    /// <summary>FT-04</summary>
	{attribute 'OPC.UA.DA' := '1'}  				                
	{attribute 'OPC.UA.DA.Access' := '1'}  					                
	product_condenser_pump_outlet_liquid_flow							: REAL;
    /// <summary>FT-04</summary>
	{attribute 'OPC.UA.DA' := '1'}  				                
	{attribute 'OPC.UA.DA.Access' := '1'}  				                
	product_condenser_pump_outlet_liquid_flow_error				AT %I*	: BOOL;
    /// <summary>product condenser pump liquid flow</summary>
	FT_04														AT %I*	: INT;
	
    /// <summary>FT-05</summary>
	{attribute 'OPC.UA.DA' := '1'}  				                
	{attribute 'OPC.UA.DA.Access' := '1'}  					                
	tap_water_to_boiler_flow											: REAL;
	/// <summary>FT-05</summary>
	{attribute 'OPC.UA.DA' := '1'}  				                
	{attribute 'OPC.UA.DA.Access' := '1'}  					                
	tap_water_to_boiler_flow_total										: REAL;
	/// <summary>FT-05</summary>
	{attribute 'OPC.UA.DA' := '1'}  				                					                
	tap_water_to_boiler_flow_total_enable								: BOOL;
    /// <summary>FT-05</summary>
	{attribute 'OPC.UA.DA' := '1'}  				                
	{attribute 'OPC.UA.DA.Access' := '1'}  				                
	tap_water_to_boiler_flow_error								AT %I*	: BOOL;
    /// <summary>tap water to boiler flow</summary>
	FT_05														AT %I*	: INT;

    /// <summary>FT-06</summary>
	{attribute 'OPC.UA.DA' := '1'}  				                
	{attribute 'OPC.UA.DA.Access' := '1'}  					                
	steam_header_flow													: REAL;
	{attribute 'OPC.UA.DA' := '1'}  				                
	{attribute 'OPC.UA.DA.Access' := '1'}
	steam_header_volume  												: REAL;
	 /// <summary>FT-06</summary>
	{attribute 'OPC.UA.DA' := '1'}  				                
	{attribute 'OPC.UA.DA.Access' := '1'}
	steam_header_volume_total 											: REAL;
	  /// <summary>FT-06</summary>
	{attribute 'OPC.UA.DA' := '1'} 
	steam_header_volume_total_enable 									: BOOL;
    /// <summary>FT-06</summary>
	{attribute 'OPC.UA.DA' := '1'}  				                
	{attribute 'OPC.UA.DA.Access' := '1'}  				                
	steam_header_flow_error										AT %I*	: BOOL;
    /// <summary>steam header flow</summary>
	FT_06														AT %I*	: INT;

    /// <summary>FT-07</summary>
	{attribute 'OPC.UA.DA' := '1'}  				                
	{attribute 'OPC.UA.DA.Access' := '1'}  					                
	condensate_collection_tank_flow										: REAL;
    /// <summary>FT-07</summary>
	{attribute 'OPC.UA.DA' := '1'}  				                
	{attribute 'OPC.UA.DA.Access' := '1'}  				                
	condensate_collection_tank_flow_error						AT %I*	: BOOL;
    /// <summary>condensate collection tank flow</summary>
	FT_07														AT %I*	: INT;

    /// <summary>AT-08</summary>
	{attribute 'OPC.UA.DA' := '1'}  				                
	{attribute 'OPC.UA.DA.Access' := '1'}  				                
	weather_wind_speed													: REAL;
    /// <summary>AT-08</summary>                        
	{attribute 'OPC.UA.DA' := '1'}  				                
	{attribute 'OPC.UA.DA.Access' := '1'}  				            
	weather_wind_speed_error									AT %I*	: BOOL;
    /// <summary>weather wind speed</summary>
	AT_08														AT %I*	: INT;

    /// <summary>LT-01</summary>
	{attribute 'OPC.UA.DA' := '1'}  				                
	{attribute 'OPC.UA.DA.Access' := '1'}  					                
	product_condensate_drum_level										: REAL;
    /// <summary>LT-01</summary>
	{attribute 'OPC.UA.DA' := '1'}  				                
	{attribute 'OPC.UA.DA.Access' := '1'}  				                
	product_condensate_drum_level_error							AT %I*	: BOOL;
    /// <summary>product condensate drum level</summary>
	LT_01														AT %I*	: INT;

    /// <summary>LT-02</summary>
	{attribute 'OPC.UA.DA' := '1'}  				                
	{attribute 'OPC.UA.DA.Access' := '1'}  					                
	condensate_collection_tank_level									: REAL;
    /// <summary>LT-02</summary>
	{attribute 'OPC.UA.DA' := '1'}  				                
	{attribute 'OPC.UA.DA.Access' := '1'}  				                
	condensate_collection_tank_level_error						AT %I*	: BOOL;
    /// <summary>condensate collection tank flow</summary>
	LT_02														AT %I*	: INT;

    /// <summary>PT-01</summary>
	{attribute 'OPC.UA.DA' := '1'}  				                
	{attribute 'OPC.UA.DA.Access' := '1'}  				                
	dead_air_line_pres													: REAL;
    /// <summary>PT-01</summary>
	{attribute 'OPC.UA.DA' := '1'}  				                
	{attribute 'OPC.UA.DA.Access' := '1'}  				                
	dead_air_line_pres_error									AT %I*	: BOOL;
    /// <summary>dead air line pres</summary>
	PT_01														AT %I*	: INT;
	
    /// <summary>PT-02</summary>
	{attribute 'OPC.UA.DA' := '1'}  				                
	{attribute 'OPC.UA.DA.Access' := '1'}  				                
	purge_product_line_pres												: REAL;
    /// <summary>PT-02</summary>
	{attribute 'OPC.UA.DA' := '1'}  				                
	{attribute 'OPC.UA.DA.Access' := '1'}  				                
	purge_product_line_pres_error								AT %I*	: BOOL;
    /// <summary>product line pres</summary>
	PT_02														AT %I*	: INT;

    /// <summary>PT-03</summary>
	{attribute 'OPC.UA.DA' := '1'}  				                
	{attribute 'OPC.UA.DA.Access' := '1'}  				                
	pre_condenser_line_pres												: REAL;
    /// <summary>PT-03</summary>
	{attribute 'OPC.UA.DA' := '1'}  				                
	{attribute 'OPC.UA.DA.Access' := '1'}  				                
	pre_condenser_line_pres_error								AT %I*	: BOOL;
    /// <summary>pre condenser line pres</summary>
	PT_03														AT %I*	: INT;

    /// <summary>PT-04</summary>
	{attribute 'OPC.UA.DA' := '1'}  				                
	{attribute 'OPC.UA.DA.Access' := '1'}  				                
	post_condenser_line_pres											: REAL;
    /// <summary>PT-04</summary>
	{attribute 'OPC.UA.DA' := '1'}  				                
	{attribute 'OPC.UA.DA.Access' := '1'}  				                
	post_condenser_line_pres_error								AT %I*	: BOOL;
    /// <summary>post condenser line pres</summary>
	PT_04														AT %I*	: INT;

    /// <summary>PT-05</summary>
	{attribute 'OPC.UA.DA' := '1'}  				                
	{attribute 'OPC.UA.DA.Access' := '1'}  				                
	product_vacuum_pres													: REAL;
    /// <summary>PT-05</summary>
	{attribute 'OPC.UA.DA' := '1'}  				                
	{attribute 'OPC.UA.DA.Access' := '1'}  				                
	product_vacuum_pres_error									AT %I*	: BOOL;
    /// <summary>product vacuum pres</summary>
	PT_05														AT %I*	: INT;

    /// <summary>P02-PT-01</summary>
	{attribute 'OPC.UA.DA' := '1'}  				                
	{attribute 'OPC.UA.DA.Access' := '1'}  				                
	product_vacuum_inlet_pres											: REAL;
    /// <summary>P02-PT-01</summary>
	{attribute 'OPC.UA.DA' := '1'}  				                
	{attribute 'OPC.UA.DA.Access' := '1'}  				                
	product_vacuum_inlet_pres_error								AT %I*	: BOOL;
	
	/// <summary>PT-06</summary>
	{attribute 'OPC.UA.DA' := '1'}  				                
	{attribute 'OPC.UA.DA.Access' := '1'}  				                
	product_outlet_pres													: REAL;
    /// <summary>PT-06</summary>
	{attribute 'OPC.UA.DA' := '1'}  				                
	{attribute 'OPC.UA.DA.Access' := '1'}  				                
	product_outlet_pres_error									AT %I*	: BOOL;
    /// <summary>product outlet pres</summary>
	PT_06														AT %I*	: INT;

    /// <summary>PT-07</summary>
	{attribute 'OPC.UA.DA' := '1'}  				                
	{attribute 'OPC.UA.DA.Access' := '1'}  				                
	boiler_outlet_pres													: REAL;
    /// <summary>PT-07</summary>
	{attribute 'OPC.UA.DA' := '1'}  				                
	{attribute 'OPC.UA.DA.Access' := '1'}  				                
	boiler_outlet_pres_error									AT %I*	: BOOL;
    /// <summary>boiler outlet pres</summary>
	PT_07														AT %I*	: INT;

    /// <summary>PT-08</summary>
	{attribute 'OPC.UA.DA' := '1'}  				                
	{attribute 'OPC.UA.DA.Access' := '1'}  				                
	instrument_air_comp_pres											: REAL;
    /// <summary>PT-08</summary>
	{attribute 'OPC.UA.DA' := '1'}  				                
	{attribute 'OPC.UA.DA.Access' := '1'}  				                
	instrument_air_comp_pres_error								AT %I*	: BOOL;
    /// <summary>instrument air comp pres</summary>
	PT_08														AT %I*	: INT;

    /// <summary>PT-09</summary>
	{attribute 'OPC.UA.DA' := '1'}  				                
	{attribute 'OPC.UA.DA.Access' := '1'}  				                
	weather_pres														: REAL;
    /// <summary>PT-09</summary>                        
	{attribute 'OPC.UA.DA' := '1'}  				                
	{attribute 'OPC.UA.DA.Access' := '1'}  				            
	weather_pres_error											AT %I*	: BOOL;
    /// <summary>weather pres</summary>
	PT_09														AT %I*	: INT;


    /// <summary>TT-01</summary>
	{attribute 'OPC.UA.DA' := '1'}  				                
	{attribute 'OPC.UA.DA.Access' := '1'}  				                
	purge_product_line_temp												: REAL;
    /// <summary>TT-01</summary>
	{attribute 'OPC.UA.DA' := '1'}  				                
	{attribute 'OPC.UA.DA.Access' := '1'}  				                
	purge_product_line_temp_error								AT %I*	: BOOL;
    /// <summary>purge product line temp</summary>
	TT_01														AT %I*	: INT;

    /// <summary>TT-02</summary>
	{attribute 'OPC.UA.DA' := '1'}  				                
	{attribute 'OPC.UA.DA.Access' := '1'}  				                
	pre_condenser_line_temp												: REAL;
    /// <summary>TT-02</summary>
	{attribute 'OPC.UA.DA' := '1'}  				                
	{attribute 'OPC.UA.DA.Access' := '1'}  				                
	pre_condenser_line_temp_error								AT %I*	: BOOL;
    /// <summary>pre condenser line temp</summary>
	TT_02														AT %I*	: INT;

    /// <summary>TT-03</summary>
	{attribute 'OPC.UA.DA' := '1'}  				                
	{attribute 'OPC.UA.DA.Access' := '1'}  				                
	post_condenser_line_temp												: REAL;
    /// <summary>TT-03</summary>
	{attribute 'OPC.UA.DA' := '1'}  				                
	{attribute 'OPC.UA.DA.Access' := '1'}  				                
	post_condenser_line_temp_error								AT %I*	: BOOL;
    /// <summary>purge product line temp</summary>
	TT_03														AT %I*	: INT;

    /// <summary>TT-04</summary>
	{attribute 'OPC.UA.DA' := '1'}  				                
	{attribute 'OPC.UA.DA.Access' := '1'}  				                
	product_outlet_temp													: REAL;
    /// <summary>TT-04</summary>
	{attribute 'OPC.UA.DA' := '1'}  				                
	{attribute 'OPC.UA.DA.Access' := '1'}  				                
	product_outlet_temp_error									AT %I*	: BOOL;
    /// <summary>product outlet temp</summary>
	TT_04														AT %I*	: INT;

    /// <summary>TT-05</summary>
	{attribute 'OPC.UA.DA' := '1'}  				                
	{attribute 'OPC.UA.DA.Access' := '1'}  				                
	product_condenser_pump_outlet_temp									: REAL;
    /// <summary>TT-05</summary>
	{attribute 'OPC.UA.DA' := '1'}  				                
	{attribute 'OPC.UA.DA.Access' := '1'}  				                
	product_condenser_pump_outlet_temp_error					AT %I*	: BOOL;
    /// <summary>product condenser pump outlet temp</summary>
	TT_05														AT %I*	: INT;

    /// <summary>TT-06</summary>
	{attribute 'OPC.UA.DA' := '1'}  				                
	{attribute 'OPC.UA.DA.Access' := '1'}  				                
	boiler_outlet_temp													: REAL;
    /// <summary>TT-06</summary>
	{attribute 'OPC.UA.DA' := '1'}  				                
	{attribute 'OPC.UA.DA.Access' := '1'}  				                
	boiler_outlet_temp_error									AT %I*	: BOOL;
    /// <summary>boiler outlet temp</summary>
	TT_06														AT %I*	: INT;

    /// <summary>TT-07</summary>
	{attribute 'OPC.UA.DA' := '1'}  				                
	{attribute 'OPC.UA.DA.Access' := '1'}  				                
	condensate_collection_tank_temp										: REAL;
    /// <summary>TT-07</summary>
	{attribute 'OPC.UA.DA' := '1'}  				                
	{attribute 'OPC.UA.DA.Access' := '1'}  				                
	condensate_collection_tank_temp_error						AT %I*	: BOOL;
    /// <summary>condensate collection tank temp</summary>
	TT_07														AT %I*	: INT;

    /// <summary>TT-08</summary>
	{attribute 'OPC.UA.DA' := '1'}  				                
	{attribute 'OPC.UA.DA.Access' := '1'}  				                
	condensate_collection_tank_outlet_line_temp							: REAL;
    /// <summary>TT-08</summary>
	{attribute 'OPC.UA.DA' := '1'}  				                
	{attribute 'OPC.UA.DA.Access' := '1'}  				                
	condensate_collection_tank_outlet_line_temp_error			AT %I*	: BOOL;
    /// <summary>condensate collection tank outlet temp</summary>
	TT_08														AT %I*	: INT;

    /// <summary>TT-09</summary>
	{attribute 'OPC.UA.DA' := '1'}  				                
	{attribute 'OPC.UA.DA.Access' := '1'}  				                
	instrument_air_comp_temp											: REAL;
    /// <summary>TT-09</summary>
	{attribute 'OPC.UA.DA' := '1'}  				                
	{attribute 'OPC.UA.DA.Access' := '1'}  				                
	instrument_air_comp_temp_error								AT %I*	: BOOL;
    /// <summary>instrument air comp temp</summary>
	TT_09														AT %I*	: INT;

    /// <summary>TT-10</summary>
	{attribute 'OPC.UA.DA' := '1'}  				                
	{attribute 'OPC.UA.DA.Access' := '1'}  				                
	weather_temp														: REAL;
    /// <summary>TT-10</summary>
	{attribute 'OPC.UA.DA' := '1'}  				                
	{attribute 'OPC.UA.DA.Access' := '1'}  				                
	weather_temp_error											AT %I*	: BOOL;
    /// <summary>instrument air comp temp</summary>
	TT_10														AT %I*	: INT;


    /// <summary>NT-01</summary>
	{attribute 'OPC.UA.DA' := '1'}  				                
	{attribute 'OPC.UA.DA.Access' := '1'}  				                
	weather_noise_level													: REAL;
    /// <summary>NT-01</summary>
	{attribute 'OPC.UA.DA' := '1'}  				                
	{attribute 'OPC.UA.DA.Access' := '1'}  				                
	weather_noise_level_error									AT %I*	: BOOL;
    /// <summary>weather noise level</summary>
	NT_01														AT %I*	: INT;

	
    /// <summary>WDT-01</summary>
	{attribute 'OPC.UA.DA' := '1'}  				                
	{attribute 'OPC.UA.DA.Access' := '1'}  				                
	weather_wind_direction												: REAL;
    /// <summary>WDT-01</summary>
	{attribute 'OPC.UA.DA' := '1'}  				                
	{attribute 'OPC.UA.DA.Access' := '1'}  				                
	weather_wind_direction_error								AT %I*	: BOOL;
    /// <summary>weather wind direction</summary>
	WDT_01														AT %I*	: INT;

	
    /// <summary>XV-01</summary>
	{attribute 'OPC.UA.DA' := '1'}  				                
	cooling_line_pre_condenser_valve									: BOOL;
    /// <summary>XV-01</summary>
	{attribute 'OPC.UA.DA' := '1'}  				                
	{attribute 'OPC.UA.DA.Access' := '1'}  				                
	cooling_line_pre_condenser_valve_open_cmd_status					: BOOL;
    /// <summary>XV-01</summary>
	{attribute 'OPC.UA.DA' := '1'}  				                
	{attribute 'OPC.UA.DA.Access' := '1'}  				                
	cooling_line_pre_condenser_valve_open						AT %I*	: BOOL;
    /// <summary>XV-01</summary>
	{attribute 'OPC.UA.DA' := '1'}  				                
	{attribute 'OPC.UA.DA.Access' := '1'}  				                
	cooling_line_pre_condenser_valve_closed						AT %I*	: BOOL;
    /// <summary>cooling line pre condenser valve</summary>
	XV_01														AT %Q*	: BOOL;
	
    /// <summary>XV-02</summary>
	{attribute 'OPC.UA.DA' := '1'}  				                
	purge_product_pre_condenser_valve									: BOOL;
    /// <summary>XV-02</summary>
	{attribute 'OPC.UA.DA' := '1'}  				                
	{attribute 'OPC.UA.DA.Access' := '1'}  				                
	purge_product_pre_condenser_valve_open_cmd_status					: BOOL;
    /// <summary>XV-02</summary>
	{attribute 'OPC.UA.DA' := '1'}  				                
	{attribute 'OPC.UA.DA.Access' := '1'}  				                
	purge_product_pre_condenser_valve_open						AT %I*	: BOOL;
    /// <summary>XV-02</summary>
	{attribute 'OPC.UA.DA' := '1'}  				                
	{attribute 'OPC.UA.DA.Access' := '1'}  				                
	purge_product_pre_condenser_valve_closed					AT %I*	: BOOL;
    /// <summary>purge product pre condenser valve</summary>
	XV_02														AT %Q*	: BOOL;
	
    /// <summary>XV-03</summary>
	{attribute 'OPC.UA.DA' := '1'}  				                
	product_vacuum_pump_isolation_valve									: BOOL;
    /// <summary>XV-03</summary>
	{attribute 'OPC.UA.DA' := '1'}  				                
	{attribute 'OPC.UA.DA.Access' := '1'}  				                
	product_vacuum_pump_isolation_valve_open_cmd_status					: BOOL;
    /// <summary>XV-03</summary>
	{attribute 'OPC.UA.DA' := '1'}  				                
	{attribute 'OPC.UA.DA.Access' := '1'}  				                
	product_vacuum_pump_isolation_valve_open					AT %I*	: BOOL;
    /// <summary>XV-03</summary>
	{attribute 'OPC.UA.DA' := '1'}  				                
	{attribute 'OPC.UA.DA.Access' := '1'}  				                
	product_vacuum_pump_isolation_valve_closed					AT %I*	: BOOL;
    /// <summary>product vacuum pump isolation valve</summary>
	XV_03														AT %Q*	: BOOL;
	
    /// <summary>XV-04</summary>
	{attribute 'OPC.UA.DA' := '1'}  				                
	product_vacuum_bypass_valve											: BOOL;
    /// <summary>XV-04</summary>
	{attribute 'OPC.UA.DA' := '1'}  				                
	{attribute 'OPC.UA.DA.Access' := '1'}  				                
	product_vacuum_bypass_valve_open_cmd_status							: BOOL;
    /// <summary>XV-04</summary>
	{attribute 'OPC.UA.DA' := '1'}  				                
	{attribute 'OPC.UA.DA.Access' := '1'}  				                
	product_vacuum_bypass_valve_open							AT %I*	: BOOL;
    /// <summary>XV-04</summary>
	{attribute 'OPC.UA.DA' := '1'}  				                
	{attribute 'OPC.UA.DA.Access' := '1'}  				                
	product_vacuum_bypass_valve_closed							AT %I*	: BOOL;
    /// <summary>product vacuum bypass valve</summary>
	XV_04														AT %Q*	: BOOL;
	
    /// <summary>XV-05</summary>
	{attribute 'OPC.UA.DA' := '1'}  				                
	product_vacuum_outlet_isolation_valve								: BOOL;
    /// <summary>XV-05</summary>
	{attribute 'OPC.UA.DA' := '1'}  				                
	{attribute 'OPC.UA.DA.Access' := '1'}  				                
	product_vacuum_outlet_isolation_valve_open_cmd_status				: BOOL;
    /// <summary>XV-05</summary>
	{attribute 'OPC.UA.DA' := '1'}  				                
	{attribute 'OPC.UA.DA.Access' := '1'}  				                
	product_vacuum_outlet_isolation_valve_open					AT %I*	: BOOL;
    /// <summary>XV-05</summary>
	{attribute 'OPC.UA.DA' := '1'}  				                
	{attribute 'OPC.UA.DA.Access' := '1'}  				                
	product_vacuum_outlet_isolation_valve_closed				AT %I*	: BOOL;
    /// <summary>product vacuum outlet isolation valve</summary>
	XV_05														AT %Q*	: BOOL;
	
    /// <summary>XV-06</summary>
	{attribute 'OPC.UA.DA' := '1'}  				                
	product_condensate_drain_valve										: BOOL;
    /// <summary>XV-06</summary>
	{attribute 'OPC.UA.DA' := '1'}  				                
	{attribute 'OPC.UA.DA.Access' := '1'}  				                
	product_condensate_drain_valve_open_cmd_status						: BOOL;
    /// <summary>XV-06</summary>
	{attribute 'OPC.UA.DA' := '1'}  				                
	{attribute 'OPC.UA.DA.Access' := '1'}  				                
	product_condensate_drain_valve_open							AT %I*	: BOOL;
    /// <summary>XV-06</summary>
	{attribute 'OPC.UA.DA' := '1'}  				                
	{attribute 'OPC.UA.DA.Access' := '1'}  				                
	product_condensate_drain_valve_closed						AT %I*	: BOOL;
    /// <summary>product condensate drain valve</summary>
	XV_06														AT %Q*	: BOOL;
	
    /// <summary>XV-08</summary>
	{attribute 'OPC.UA.DA' := '1'}  				                
	steam_bypass_valve													: BOOL;
    /// <summary>XV-08</summary>
	{attribute 'OPC.UA.DA' := '1'}  				                
	{attribute 'OPC.UA.DA.Access' := '1'}  				                
	steam_bypass_valve_open_cmd_status									: BOOL;
    /// <summary>XV-08</summary>
	{attribute 'OPC.UA.DA' := '1'}  				                
	{attribute 'OPC.UA.DA.Access' := '1'}  				                
	steam_bypass_valve_open										AT %I*	: BOOL;
    /// <summary>XV-08</summary>
	{attribute 'OPC.UA.DA' := '1'}  				                
	{attribute 'OPC.UA.DA.Access' := '1'}  				                
	steam_bypass_valve_closed									AT %I*	: BOOL;
    /// <summary>steam bypass valve</summary>
	XV_08														AT %Q*	: BOOL;
    
	/// <summary>XV-09</summary>
	{attribute 'OPC.UA.DA' := '1'}  				                
	condensate_collection_tank_pump_outlet_valve						: BOOL;
    /// <summary>XV-09</summary>
	{attribute 'OPC.UA.DA' := '1'}  				                
	{attribute 'OPC.UA.DA.Access' := '1'}  				                
	condensate_collection_tank_pump_outlet_valve_open_cmd_status		: BOOL;
    /// <summary>XV-09</summary>
	{attribute 'OPC.UA.DA' := '1'}  				                
	{attribute 'OPC.UA.DA.Access' := '1'}  				                
	condensate_collection_tank_pump_outlet_valve_open			AT %I*	: BOOL;
    /// <summary>XV-09</summary>
	{attribute 'OPC.UA.DA' := '1'}  				                
	{attribute 'OPC.UA.DA.Access' := '1'}  				                
	condensate_collection_tank_pump_outlet_valve_closed 		AT %I*	: BOOL;
    /// <summary>condensate collection tank pump outlet valve</summary>
	XV_09														AT %Q*	: BOOL;

    /// <summary>PCV-01</summary>
	product_vacuum_backfeed_valve_open									: BOOL;
    /// <summary>PCV-01</summary>
	product_vacuum_backfeed_valve_closed								: BOOL;
    /// <summary>PCV-01</summary>
	{attribute 'OPC.UA.DA' := '1'}  				                
	product_vacuum_backfeed_valve										: REAL;
    /// <summary>PCV-01</summary>
	{attribute 'OPC.UA.DA' := '1'}  				                
	{attribute 'OPC.UA.DA.Access' := '1'}  				                
	product_vacuum_backfeed_valve_position								: REAL;
    /// <summary>PCV-01</summary>
	{attribute 'OPC.UA.DA' := '1'}  				                
	{attribute 'OPC.UA.DA.Access' := '1'}  				                
	product_vacuum_backfeed_valve_position_error				AT %I*	: BOOL;
    /// <summary>product vacuum backfeed valve</summary>
	PCV_01														AT %Q*	: INT;
    /// <summary>product vacuum backfeed valve</summary>
	{attribute 'OPC.UA.DA' := '1'}  				                
	{attribute 'OPC.UA.DA.Access' := '1'}  				                
	PCV_01_position												AT %I*	: INT;
    /// <summary>PCV-01</summary>                  	           
	{attribute 'OPC.UA.DA' := '1'}  				                
	product_vacuum_backfeed_valve_mode									: INT;			
    /// <summary>PCV-01</summary>                  	           
	{attribute 'OPC.UA.DA' := '1'}  				                
	{attribute 'OPC.UA.DA.Access' := '1'}  				                
	product_vacuum_backfeed_valve_current_mode							: INT;			
    /// <summary>PCV-01</summary>                  	           
	product_vacuum_backfeed_valve_kp									: REAL		:= 0.01; 
    /// <summary>PCV-01</summary>                  	           
	product_vacuum_backfeed_valve_ki									: REAL		:= 0.01;
    /// <summary>PCV-01</summary>                  	           
	product_vacuum_backfeed_valve_loop_time								: REAL		:= 2000;
    /// <summary>PCV-01</summary>                  	           
	product_vacuum_backfeed_valve_iband									: REAL		:= 6;
    /// <summary>PCV-01</summary>                  	           
	product_vacuum_backfeed_valve_base									: INT		:= 13110;
    /// <summary>PCV-01</summary>                  	           
	product_vacuum_backfeed_valve_base_adjust							: INT		:= 10;
	
    /// <summary>P-02</summary>
	{attribute 'OPC.UA.DA' := '1'}  				                
	product_vacuum_pump_reset											: BOOL;												// PS 04_17_24 Added for Vacuum Pump FB reset
    /// <summary>P-02</summary>
	{attribute 'OPC.UA.DA' := '1'}  				                
	product_vacuum_pump_vfd_reset										: BOOL;
	  /// <summary>P-02</summary>
	{attribute 'OPC.UA.DA' := '1'}  				                
	product_vacuum_pump_vfd_enable										: BOOL;
    /// <summary>P-02</summary>
	{attribute 'OPC.UA.DA' := '1'}  				                
	{attribute 'OPC.UA.DA.Access' := '1'}  				                
	product_vacuum_pump_vfd_enabled										: BOOL;
    /// <summary>P-02</summary>
	{attribute 'OPC.UA.DA' := '1'}  				                
	{attribute 'OPC.UA.DA.Access' := '1'}  				                
	product_vacuum_pump_vfd_error										: BOOL;
    /// <summary>P-02</summary>
	{attribute 'OPC.UA.DA' := '1'}  				                
	product_vacuum_pump_vfd												: REAL;
    /// <summary>P-02</summary>
	{attribute 'OPC.UA.DA' := '1'}  				                
    /// <summary>P-02</summary>
	product_vacuum_pump_vfd_output										: REAL;
    /// <summary>P-02</summary>
	product_vacuum_pump_vfd_control								AT %Q*	: WORD;
    /// <summary>P-02</summary>
	product_vacuum_pump_vfd_target_vel							AT %Q*	: WORD;
    /// <summary>P-02</summary>
	product_vacuum_pump_vfd_status								AT %I*	: WORD;
    /// <summary>P-02</summary>
	product_vacuum_pump_vfd_velocity							AT %I*	: WORD;

    /// <summary>product_vacuum_pump_pressure</summary>
	P02_PT_01													AT %I*	: INT;
    /// <summary>product_vacuum_pump_cooling_jacket_temp_trip_switch</summary>
	P02_TSH_1													AT %I*	: BOOL;
    /// <summary>product_vacuum_pump_exhaust_temp_trip_switch</summary>
	P02_TSH_2													AT %I*	: BOOL;
    /// <summary>product_vacuum_pump_oil_temp_trip_switch</summary>
	P02_TSH_3													AT %I*	: BOOL;
    /// <summary>product_vacuum_pump_purge_solenoid_valve</summary>
	P02_SVC_1													AT %Q*	: BOOL;
    /// <summary>product_vacuum_pump_seal_purge_valve</summary>
	P02_SVC_3													AT %Q*	: BOOL;
	product_vacuum_pump_error											: INT;
	
	
	  /// <summary>AT-04_pump</summary>
	{attribute 'OPC.UA.DA' := '1'}  				                
	product_co2_chiller_pump											: BOOL;
    /// <summary>AT-04_pump</summary>
	{attribute 'OPC.UA.DA' := '1'}  				                
	{attribute 'OPC.UA.DA.Access' := '1'}  				                
	product_co2_chiller_pump_cmd_status									: BOOL;
    /// <summary>product chiller CO2 pump</summary>
	AT_04_pump													AT %Q*	: BOOL;
    /// <summary>AT-04_chiller</summary>
	{attribute 'OPC.UA.DA' := '1'}  				                
	product_co2_chiller													: BOOL;
    /// <summary>AT-04_chiller</summary>
	{attribute 'OPC.UA.DA' := '1'}  				                
	{attribute 'OPC.UA.DA.Access' := '1'}  				                
	product_co2_chiller_cmd_status											: BOOL;
    /// <summary>productCO2 chiller</summary>
	AT_04_chiller												AT %Q*	: BOOL;
	
	
	
	{attribute 'OPC.UA.DA' := '1'}  				                
	{attribute 'OPC.UA.DA.Access' := '1'}  				                
	l1_current_480														: REAL;
	{attribute 'OPC.UA.DA' := '1'}  				                
	{attribute 'OPC.UA.DA.Access' := '1'}  				                
	l1_current_480_error										AT %I*	: BOOL;
	IT_01														AT %I*	: INT;
	{attribute 'OPC.UA.DA' := '1'}  				                
	{attribute 'OPC.UA.DA.Access' := '1'}  				                
	l2_current_480														: REAL;
	{attribute 'OPC.UA.DA' := '1'}  				                
	{attribute 'OPC.UA.DA.Access' := '1'}  				                
	l2_current_480_error										AT %I*	: BOOL;
	IT_02														AT %I*	: INT;
	{attribute 'OPC.UA.DA' := '1'}  				                
	{attribute 'OPC.UA.DA.Access' := '1'}  				                
	l3_current_480														: REAL;
	{attribute 'OPC.UA.DA' := '1'}  				                
	{attribute 'OPC.UA.DA.Access' := '1'}  				                
	l3_current_480_error										AT %I*	: BOOL;
	IT_03														AT %I*	: INT;
	
	{attribute 'OPC.UA.DA' := '1'}  				                
	{attribute 'OPC.UA.DA.Access' := '1'}  				                
	l1_voltage_480														: REAL;
	{attribute 'OPC.UA.DA' := '1'}  				                
	{attribute 'OPC.UA.DA.Access' := '1'}  				                
	l1_voltage_480_error										AT %I*	: BOOL;
	{attribute 'OPC.UA.DA' := '1'}  				                
	VT_01														AT %I*	: INT;
	{attribute 'OPC.UA.DA' := '1'}  				                
	l2_voltage_480														: REAL;
	{attribute 'OPC.UA.DA' := '1'}  				                
	{attribute 'OPC.UA.DA.Access' := '1'}  				                
	l2_voltage_480_error										AT %I*	: BOOL;
	{attribute 'OPC.UA.DA' := '1'}  				                
	VT_02														AT %I*	: INT;
	{attribute 'OPC.UA.DA' := '1'}  				                
	l3_voltage_480														: REAL;
	{attribute 'OPC.UA.DA' := '1'}  				                
	{attribute 'OPC.UA.DA.Access' := '1'}  				                
	l3_voltage_480_error										AT %I*	: BOOL;
	{attribute 'OPC.UA.DA' := '1'}  				                
	VT_03														AT %I*	: INT;
	
	{attribute 'OPC.UA.DA' := '1'}  				                
	{attribute 'OPC.UA.DA.Access' := '1'}  				                
	l1_current_208														: REAL;
	{attribute 'OPC.UA.DA' := '1'}  				                
	{attribute 'OPC.UA.DA.Access' := '1'}  				                
	l1_current_208_error										AT %I*	: BOOL;
	IT_04														AT %I*	: INT;
	{attribute 'OPC.UA.DA' := '1'}  				                
	{attribute 'OPC.UA.DA.Access' := '1'}  				                
	l2_current_208														: REAL;
	{attribute 'OPC.UA.DA' := '1'}  				                
	{attribute 'OPC.UA.DA.Access' := '1'}  				                
	l2_current_208_error										AT %I*	: BOOL;
	IT_05														AT %I*	: INT;
	{attribute 'OPC.UA.DA' := '1'}  				                
	{attribute 'OPC.UA.DA.Access' := '1'}  				                
	l3_current_208														: REAL;
	{attribute 'OPC.UA.DA' := '1'}  				                
	{attribute 'OPC.UA.DA.Access' := '1'}  				                
	l3_current_208_error										AT %I*	: BOOL;
	IT_06														AT %I*	: INT;
	
	{attribute 'OPC.UA.DA' := '1'}  				                
	{attribute 'OPC.UA.DA.Access' := '1'}  				                
	l1_voltage_208														: REAL;
	{attribute 'OPC.UA.DA' := '1'}  				                
	{attribute 'OPC.UA.DA.Access' := '1'}  				                
	l1_voltage_208_error										AT %I*	: BOOL;
	VT_04														AT %I*	: INT;
	{attribute 'OPC.UA.DA' := '1'}  				                
	{attribute 'OPC.UA.DA.Access' := '1'}  				                
	l2_voltage_208														: REAL;
	{attribute 'OPC.UA.DA' := '1'}  				                
	{attribute 'OPC.UA.DA.Access' := '1'}  				                
	l2_voltage_208_error										AT %I*	: BOOL;
	VT_05														AT %I*	: INT;
	{attribute 'OPC.UA.DA' := '1'}  				                
	{attribute 'OPC.UA.DA.Access' := '1'}  				                
	l3_voltage_208														: REAL;
	{attribute 'OPC.UA.DA' := '1'}  				                
	{attribute 'OPC.UA.DA.Access' := '1'}  				                
	l3_voltage_208_error										AT %I*	: BOOL;
	VT_06														AT %I*	: INT;
	
	{attribute 'OPC.UA.DA' := '1'}  				                
	{attribute 'OPC.UA.DA.Access' := '1'}  				                
	l1_current_boiler													: REAL;
	{attribute 'OPC.UA.DA' := '1'}  				                
	{attribute 'OPC.UA.DA.Access' := '1'}  				                
	l1_current_boiler_error										AT %I*	: BOOL;
	IT_boiler_01												AT %I*	: INT;
	{attribute 'OPC.UA.DA' := '1'}  				                
	{attribute 'OPC.UA.DA.Access' := '1'}  				                
	l2_current_boiler													: REAL;
	{attribute 'OPC.UA.DA' := '1'}  				                
	{attribute 'OPC.UA.DA.Access' := '1'}  				                
	l2_current_boiler_error										AT %I*	: BOOL;
	IT_boiler_02												AT %I*	: INT;
	{attribute 'OPC.UA.DA' := '1'}  				                
	{attribute 'OPC.UA.DA.Access' := '1'}  				                
	l3_current_boiler													: REAL;
	{attribute 'OPC.UA.DA' := '1'}  				                
	{attribute 'OPC.UA.DA.Access' := '1'}  				                
	l3_current_boiler_error										AT %I*	: BOOL;
	IT_boiler_03												AT %I*	: INT;
	
END_VAR

VAR_GLOBAL PERSISTENT
	
	/// SCALING
	
    /// <summary>AT-01</summary>
	{attribute 'OPC.UA.DA' := '1'}  				                
	dead_air_line_co2_low												: REAL;
    /// <summary>AT-01</summary>
	{attribute 'OPC.UA.DA' := '1'}  				                
	dead_air_line_co2_high												: REAL;
    /// <summary>AT-01</summary>
	{attribute 'OPC.UA.DA' := '1'}  				                
	dead_air_line_co2_min												: REAL;
    /// <summary>AT-01</summary>
	{attribute 'OPC.UA.DA' := '1'}  				                
	dead_air_line_co2_offset											: REAL;
	
    /// <summary>AT-02</summary>
	{attribute 'OPC.UA.DA' := '1'}  				                
	product_outlet_co2_low												: REAL;
    /// <summary>AT-02</summary>
	{attribute 'OPC.UA.DA' := '1'}  				                
	product_outlet_co2_high												: REAL;
    /// <summary>AT-02</summary>
	{attribute 'OPC.UA.DA' := '1'}  				                
	product_outlet_co2_min												: REAL;
    /// <summary>AT-02</summary>
	{attribute 'OPC.UA.DA' := '1'}  				                
	product_outlet_co2_offset											: REAL;
	
	/// <summary>AT-02</summary>
	{attribute 'OPC.UA.DA' := '1'}  				                
	product_co2sample_h2o_low											: REAL;
    /// <summary>AT-02</summary>
	{attribute 'OPC.UA.DA' := '1'}  				                
	product_co2sample_h2o_high											: REAL;
    /// <summary>AT-02</summary>
	{attribute 'OPC.UA.DA' := '1'}  				                
	product_co2sample_h2o_min											: REAL;
    /// <summary>AT-02</summary>
	{attribute 'OPC.UA.DA' := '1'}  				                
	product_co2sample_h2o_offset										: REAL;
	
	
    /// <summary>AT-07</summary>
	{attribute 'OPC.UA.DA' := '1'}  				                
	product_outlet_h2o_low												: REAL;
    /// <summary>AT-07</summary>
	{attribute 'OPC.UA.DA' := '1'}  				                
	product_outlet_h2o_high												: REAL;
    /// <summary>AT-07</summary>
	{attribute 'OPC.UA.DA' := '1'}  				                
	product_outlet_h2o_min												: REAL;
    /// <summary>AT-07</summary>
	{attribute 'OPC.UA.DA' := '1'}  				                
	product_outlet_h2o_offset											: REAL;
	
	
	 /// <summary>AT-07</summary>
	{attribute 'OPC.UA.DA' := '1'}  				                
	product_outlet_temperature_low										: REAL;
    /// <summary>AT-07</summary>
	{attribute 'OPC.UA.DA' := '1'}  				                
	product_outlet_temperature_high										: REAL;
    /// <summary>AT-07</summary>
	{attribute 'OPC.UA.DA' := '1'}  				                
	product_outlet_temperature_min										: REAL;
    /// <summary>AT-07</summary>
	{attribute 'OPC.UA.DA' := '1'}  				                
	product_outlet_temperature_offset									: REAL;
	
    /// <summary>AT-03</summary>
	{attribute 'OPC.UA.DA' := '1'}  				                
	product_outlet_o2_low												: REAL;
    /// <summary>AT-03</summary>
	{attribute 'OPC.UA.DA' := '1'}  				                
	product_outlet_o2_high												: REAL;
    /// <summary>AT-03</summary>
	{attribute 'OPC.UA.DA' := '1'}  				                
	product_outlet_o2_min												: REAL;
    /// <summary>AT-03</summary>
	{attribute 'OPC.UA.DA' := '1'}  				                
	product_outlet_o2_offset											: REAL;
	
    /// <summary>AT-04</summary>                        
	{attribute 'OPC.UA.DA' := '1'}  				            
	condensate_collection_tank_ph_low									: REAL;
    /// <summary>AT-04</summary>                        
	{attribute 'OPC.UA.DA' := '1'}  				            
	condensate_collection_tank_ph_high									: REAL;
    /// <summary>AT-04</summary>                        
	{attribute 'OPC.UA.DA' := '1'}  				            
	condensate_collection_tank_ph_min									: REAL;
    /// <summary>AT-04</summary>                        
	{attribute 'OPC.UA.DA' := '1'}  				            
	condensate_collection_tank_ph_offset								: REAL;

    /// <summary>AT-05</summary>                        
	{attribute 'OPC.UA.DA' := '1'}  				            
	condensate_collection_tank_o2_low									: REAL;
    /// <summary>AT-05</summary>                        
	{attribute 'OPC.UA.DA' := '1'}  				            
	condensate_collection_tank_o2_high									: REAL;
    /// <summary>AT-05</summary>                        
	{attribute 'OPC.UA.DA' := '1'}  				            
	condensate_collection_tank_o2_min									: REAL;
    /// <summary>AT-05</summary>                        
	{attribute 'OPC.UA.DA' := '1'}  				            
	condensate_collection_tank_o2_offset								: REAL;
	
    /// <summary>AT-06</summary>                        
	{attribute 'OPC.UA.DA' := '1'}  				            
	condensate_collection_tank_turbidity_low							: REAL;
    /// <summary>AT-06</summary>                        
	{attribute 'OPC.UA.DA' := '1'}  				            
	condensate_collection_tank_turbidity_high							: REAL;
    /// <summary>AT-06</summary>                        
	{attribute 'OPC.UA.DA' := '1'}  				            
	condensate_collection_tank_turbidity_min							: REAL;
    /// <summary>AT-06</summary>                        
	{attribute 'OPC.UA.DA' := '1'}  				            
	condensate_collection_tank_turbidity_offset							: REAL;
	
    /// <summary>AT-07</summary>                        
	{attribute 'OPC.UA.DA' := '1'}  				            
	weather_humidity_low												: REAL;
    /// <summary>AT-07</summary>                        
	{attribute 'OPC.UA.DA' := '1'}  				            
	weather_humidity_high												: REAL;
    /// <summary>AT-07</summary>                        
	{attribute 'OPC.UA.DA' := '1'}  				            
	weather_humidity_min												: REAL;
    /// <summary>AT-07</summary>                        
	{attribute 'OPC.UA.DA' := '1'}  				            
	weather_humidity_offset												: REAL;
	
    /// <summary>FT-01</summary>
	{attribute 'OPC.UA.DA' := '1'}  				                
	dead_air_flow_low													: REAL;
    /// <summary>FT-01</summary>
	{attribute 'OPC.UA.DA' := '1'}  				                
	dead_air_flow_high													: REAL;
    /// <summary>FT-01</summary>
	{attribute 'OPC.UA.DA' := '1'}  				                
	dead_air_flow_min													: REAL;
    /// <summary>FT-01</summary>
	{attribute 'OPC.UA.DA' := '1'}  				                
	dead_air_flow_offset												: REAL;

    /// <summary>FT-02</summary>
	{attribute 'OPC.UA.DA' := '1'}  				                
	product_outlet_volumetric_flow_low									: REAL;
    /// <summary>FT-02</summary>
	{attribute 'OPC.UA.DA' := '1'}  				                
	product_outlet_volumetric_flow_high									: REAL;
    /// <summary>FT-02</summary>
	{attribute 'OPC.UA.DA' := '1'}  				                
	product_outlet_volumetric_flow_min									: REAL;
    /// <summary>FT-02</summary>
	{attribute 'OPC.UA.DA' := '1'}  				                
	product_outlet_volumetric_flow_offset								: REAL;
	
    /// <summary>FT-03</summary>
	{attribute 'OPC.UA.DA' := '1'}  				                
	product_outlet_mass_flow_low										: REAL;
    /// <summary>FT-03</summary>
	{attribute 'OPC.UA.DA' := '1'}  				                
	product_outlet_mass_flow_high										: REAL;
    /// <summary>FT-03</summary>
	{attribute 'OPC.UA.DA' := '1'}  				                
	product_outlet_mass_flow_min										: REAL;
    /// <summary>FT-03</summary>
	{attribute 'OPC.UA.DA' := '1'}  				                
	product_outlet_mass_flow_offset										: REAL;
	
	

	
	
    /// <summary>FT-04</summary>
	{attribute 'OPC.UA.DA' := '1'}  				                
	product_condenser_pump_outlet_liquid_flow_low						: REAL;
    /// <summary>FT-04</summary>
	{attribute 'OPC.UA.DA' := '1'}  				                
	product_condenser_pump_outlet_liquid_flow_high						: REAL;
    /// <summary>FT-04</summary>
	{attribute 'OPC.UA.DA' := '1'}  				                
	product_condenser_pump_outlet_liquid_flow_min						: REAL;
    /// <summary>FT-04</summary>
	{attribute 'OPC.UA.DA' := '1'}  				                
	product_condenser_pump_outlet_liquid_flow_offset					: REAL;
	
    /// <summary>FT-05</summary>
	{attribute 'OPC.UA.DA' := '1'}  				                
	tap_water_to_boiler_flow_low										: REAL;
    /// <summary>FT-05</summary>
	{attribute 'OPC.UA.DA' := '1'}  				                
	tap_water_to_boiler_flow_high										: REAL;
    /// <summary>FT-05</summary>
	{attribute 'OPC.UA.DA' := '1'}  				                
	tap_water_to_boiler_flow_min										: REAL;
    /// <summary>FT-05</summary>
	{attribute 'OPC.UA.DA' := '1'}  				                
	tap_water_to_boiler_flow_offset										: REAL;

    /// <summary>FT-07</summary>
	{attribute 'OPC.UA.DA' := '1'}  				                
	condensate_collection_tank_flow_low									: REAL;
    /// <summary>FT-07</summary>
	{attribute 'OPC.UA.DA' := '1'}  				                
	condensate_collection_tank_flow_high								: REAL;
    /// <summary>FT-07</summary>
	{attribute 'OPC.UA.DA' := '1'}  				                
	condensate_collection_tank_flow_min									: REAL;
    /// <summary>FT-07</summary>
	{attribute 'OPC.UA.DA' := '1'}  				                
	condensate_collection_tank_flow_offset								: REAL;
	
    /// <summary>AT-08</summary>                        
	{attribute 'OPC.UA.DA' := '1'}  				            
	weather_wind_speed_low												: REAL;
    /// <summary>AT-08</summary>                        
	{attribute 'OPC.UA.DA' := '1'}  				            
	weather_wind_speed_high												: REAL;
    /// <summary>AT-08</summary>                        
	{attribute 'OPC.UA.DA' := '1'}  				            
	weather_wind_speed_min												: REAL;
    /// <summary>AT-08</summary>                        
	{attribute 'OPC.UA.DA' := '1'}  				            
	weather_wind_speed_offset											: REAL;
	
    /// <summary>LT-01</summary>
	{attribute 'OPC.UA.DA' := '1'}  				                
	product_condensate_drum_level_low									: REAL;
    /// <summary>LT-01</summary>
	{attribute 'OPC.UA.DA' := '1'}  				                
	product_condensate_drum_level_high									: REAL;
    /// <summary>LT-01</summary>
	{attribute 'OPC.UA.DA' := '1'}  				                
	product_condensate_drum_level_min									: REAL;
    /// <summary>LT-01</summary>
	{attribute 'OPC.UA.DA' := '1'}  				                
	product_condensate_drum_level_offset								: REAL;
	
    /// <summary>LT-02</summary>
	{attribute 'OPC.UA.DA' := '1'}  				                
	condensate_collection_tank_level_low								: REAL;
    /// <summary>LT-02</summary>
	{attribute 'OPC.UA.DA' := '1'}  				                
	condensate_collection_tank_level_high								: REAL;
    /// <summary>LT-02</summary>
	{attribute 'OPC.UA.DA' := '1'}  				                
	condensate_collection_tank_level_min								: REAL;
    /// <summary>LT-02</summary>
	{attribute 'OPC.UA.DA' := '1'}  				                
	condensate_collection_tank_level_offset								: REAL;
	
    /// <summary>PT-01</summary>
	{attribute 'OPC.UA.DA' := '1'}  				                
	dead_air_line_pres_low												: REAL;
    /// <summary>PT-01</summary>
	{attribute 'OPC.UA.DA' := '1'}  				                
	dead_air_line_pres_high												: REAL;
    /// <summary>PT-01</summary>
	{attribute 'OPC.UA.DA' := '1'}  				                
	dead_air_line_pres_min												: REAL;
    /// <summary>PT-01</summary>
	{attribute 'OPC.UA.DA' := '1'}  				                
	dead_air_line_pres_offset											: REAL;

    /// <summary>FT-06</summary>
	{attribute 'OPC.UA.DA' := '1'}  				                
	steam_header_flow_low												: REAL;
    /// <summary>FT-06</summary>
	{attribute 'OPC.UA.DA' := '1'}  				                
	steam_header_flow_high												: REAL;
    /// <summary>FT-06</summary>
	{attribute 'OPC.UA.DA' := '1'}  				                
	steam_header_flow_min												: REAL;
    /// <summary>FT-06</summary>
	{attribute 'OPC.UA.DA' := '1'}  				                
	steam_header_flow_offset											: REAL;
	
    /// <summary>PT-02</summary>
	{attribute 'OPC.UA.DA' := '1'}  				                
	purge_product_line_pres_low											: REAL;
    /// <summary>PT-02</summary>
	{attribute 'OPC.UA.DA' := '1'}  				                
	purge_product_line_pres_high										: REAL;
    /// <summary>PT-02</summary>
	{attribute 'OPC.UA.DA' := '1'}  				                
	purge_product_line_pres_min											: REAL;
    /// <summary>PT-02</summary>
	{attribute 'OPC.UA.DA' := '1'}  				                
	purge_product_line_pres_offset										: REAL;
	
    /// <summary>PT-03</summary>
	{attribute 'OPC.UA.DA' := '1'}  				                
	pre_condenser_line_pres_low											: REAL;
    /// <summary>PT-03</summary>
	{attribute 'OPC.UA.DA' := '1'}  				                
	pre_condenser_line_pres_high										: REAL;
    /// <summary>PT-03</summary>
	{attribute 'OPC.UA.DA' := '1'}  				                
	pre_condenser_line_pres_min											: REAL;
    /// <summary>PT-03</summary>
	{attribute 'OPC.UA.DA' := '1'}  				                
	pre_condenser_line_pres_offset										: REAL;

    /// <summary>PT-04</summary>
	{attribute 'OPC.UA.DA' := '1'}  				                
	post_condenser_line_pres_low										: REAL;
    /// <summary>PT-04</summary>
	{attribute 'OPC.UA.DA' := '1'}  				                
	post_condenser_line_pres_high										: REAL;
    /// <summary>PT-04</summary>
	{attribute 'OPC.UA.DA' := '1'}  				                
	post_condenser_line_pres_min										: REAL;
    /// <summary>PT-04</summary>
	{attribute 'OPC.UA.DA' := '1'}  				                
	post_condenser_line_pres_offset										: REAL;
	
    /// <summary>PT-05</summary>
	{attribute 'OPC.UA.DA' := '1'}  				                
	product_vacuum_pres_low												: REAL;
    /// <summary>PT-05</summary>
	{attribute 'OPC.UA.DA' := '1'}  				                
	product_vacuum_pres_high											: REAL;
    /// <summary>PT-05</summary>
	{attribute 'OPC.UA.DA' := '1'}  				                
	product_vacuum_pres_min												: REAL;
    /// <summary>PT-05</summary>
	{attribute 'OPC.UA.DA' := '1'}  				                
	product_vacuum_pres_offset											: REAL;
	
    /// <summary>P02-PT-01</summary>
	{attribute 'OPC.UA.DA' := '1'}  				                
	product_vacuum_inlet_pres_low										: REAL;
    /// <summary>P02-PT-01</summary>
	{attribute 'OPC.UA.DA' := '1'}  				                
	product_vacuum_inlet_pres_high										: REAL;
    /// <summary>P02-PT-01</summary>
	{attribute 'OPC.UA.DA' := '1'}  				                
	product_vacuum_inlet_pres_min										: REAL;
    /// <summary>P02-PT-01</summary>
	{attribute 'OPC.UA.DA' := '1'}  				                
	product_vacuum_inlet_pres_offset									: REAL;
	
    /// <summary>PT-06</summary>
	{attribute 'OPC.UA.DA' := '1'}  				                
	product_outlet_pres_low												: REAL;
    /// <summary>PT-06</summary>
	{attribute 'OPC.UA.DA' := '1'}  				                
	product_outlet_pres_high											: REAL;
    /// <summary>PT-06</summary>
	{attribute 'OPC.UA.DA' := '1'}  				                
	product_outlet_pres_min												: REAL;
    /// <summary>PT-06</summary>
	{attribute 'OPC.UA.DA' := '1'}  				                
	product_outlet_pres_offset											: REAL;

    /// <summary>PT-07</summary>
	{attribute 'OPC.UA.DA' := '1'}  				                
	boiler_outlet_pres_low												: REAL;
    /// <summary>PT-07</summary>
	{attribute 'OPC.UA.DA' := '1'}  				                
	boiler_outlet_pres_high												: REAL;
    /// <summary>PT-07</summary>
	{attribute 'OPC.UA.DA' := '1'}  				                
	boiler_outlet_pres_min												: REAL;
    /// <summary>PT-07</summary>
	{attribute 'OPC.UA.DA' := '1'}  				                
	boiler_outlet_pres_offset											: REAL;
	
    /// <summary>PT-08</summary>
	{attribute 'OPC.UA.DA' := '1'}  				                
	instrument_air_comp_pres_low										: REAL;
    /// <summary>PT-08</summary>
	{attribute 'OPC.UA.DA' := '1'}  				                
	instrument_air_comp_pres_high										: REAL;
    /// <summary>PT-08</summary>
	{attribute 'OPC.UA.DA' := '1'}  				                
	instrument_air_comp_pres_min										: REAL;
    /// <summary>PT-08</summary>
	{attribute 'OPC.UA.DA' := '1'}  				                
	instrument_air_comp_pres_offset										: REAL;
	
    /// <summary>PT-09</summary>                        
	{attribute 'OPC.UA.DA' := '1'}  				            
	weather_pres_low													: REAL;
    /// <summary>PT-09</summary>                        
	{attribute 'OPC.UA.DA' := '1'}  				            
	weather_pres_high													: REAL;
    /// <summary>PT-09</summary>                        
	{attribute 'OPC.UA.DA' := '1'}  				            
	weather_pres_min													: REAL;
    /// <summary>PT-09</summary>                        
	{attribute 'OPC.UA.DA' := '1'}  				            
	weather_pres_offset													: REAL;

    /// <summary>TT-01</summary>
	{attribute 'OPC.UA.DA' := '1'}  				                
	purge_product_line_temp_offset										: REAL;
	
    /// <summary>TT-02</summary>
	{attribute 'OPC.UA.DA' := '1'}  				                
	pre_condenser_line_temp_offset										: REAL;
	
    /// <summary>TT-03</summary>
	{attribute 'OPC.UA.DA' := '1'}  				                
	post_condenser_line_temp_offset										: REAL;
	
    /// <summary>TT-04</summary>
	{attribute 'OPC.UA.DA' := '1'}  				                
	product_outlet_temp_offset											: REAL;
	
    /// <summary>TT-05</summary>
	{attribute 'OPC.UA.DA' := '1'}  				                
	product_condenser_pump_outlet_temp_offset							: REAL;
	
    /// <summary>TT-06</summary>
	{attribute 'OPC.UA.DA' := '1'}  				                
	boiler_outlet_temp_offset											: REAL;
	
    /// <summary>TT-07</summary>
	{attribute 'OPC.UA.DA' := '1'}  				                
	condensate_collection_tank_temp_offset								: REAL;

	    /// <summary>TT-08</summary>
	{attribute 'OPC.UA.DA' := '1'}  				                
	condensate_collection_tank_outlet_line_temp_offset					: REAL;
	
    /// <summary>TT-09</summary>
	{attribute 'OPC.UA.DA' := '1'}  				                
	instrument_air_comp_temp_offset										: REAL;
	
    /// <summary>TT-10</summary>
	{attribute 'OPC.UA.DA' := '1'}  				                
	weather_temp_offset													: REAL;

	
	/// SET POINTS
	
	{attribute 'OPC.UA.DA' := '1'}  				                
	SP_acceptable_high_instrument_air_pressure							: REAL;
	{attribute 'OPC.UA.DA' := '1'}  				                
	SP_acceptable_low_instrument_air_pressure							: REAL;
	{attribute 'OPC.UA.DA' := '1'}  				                
	SP_adsorb_during_steam_bypass										: BOOL;	
	{attribute 'OPC.UA.DA' := '1'}  				                
	SP_adsorb_during_warmup												: BOOL;
	{attribute 'OPC.UA.DA' := '1'}  				                
	SP_boiler_warmup_duration											: REAL;
	{attribute 'OPC.UA.DA' := '1'}  				                
	SP_condensate_collection_tank_high_level							: REAL;	
	{attribute 'OPC.UA.DA' := '1'}  				                
	SP_condensate_collection_tank_low_level								: REAL;
	{attribute 'OPC.UA.DA' := '1'}  				                
	SP_drainage_function_cutoff_pressure								: REAL;	
	{attribute 'OPC.UA.DA' := '1'}  				                
	SP_duration_to_drain_cooling_and_purge_line_in_module				: REAL;				
	{attribute 'OPC.UA.DA' := '1'}  				                
	SP_duration_to_drain_reactor_set									: REAL;	
	{attribute 'OPC.UA.DA' := '1'}  				                
	SP_maximum_duration_to_drain_reactor_set							: REAL;	
	{attribute 'OPC.UA.DA' := '1'}  				                
	SP_maximum_inlet_product_vacuum_temperature							: REAL;							// PS 04_30_24	
	{attribute 'OPC.UA.DA' := '1'}  				                
	SP_maximum_instrument_air_pressure									: REAL;		
	{attribute 'OPC.UA.DA' := '1'}  				                
	SP_maximum_instrument_air_temperature								: REAL;			
	{attribute 'OPC.UA.DA' := '1'}  				                
	SP_maximum_reasonable_sorbent_TC_reading							: REAL;
	{attribute 'OPC.UA.DA' := '1'}  				                
	SP_minimum_instrument_air_pressure									: REAL;
	{attribute 'OPC.UA.DA' := '1'}  				                
	SP_minimum_instrument_air_temperature								: REAL;			
	{attribute 'OPC.UA.DA' := '1'}  				                
	SP_minimum_reasonable_sorbent_TC_reading							: REAL;
	{attribute 'OPC.UA.DA' := '1'}  				                
	SP_minimum_steam_bypass_flow_rate									: REAL;
	{attribute 'OPC.UA.DA' := '1'}  				                
	SP_product_condensate_drum_high_level								: REAL;
	{attribute 'OPC.UA.DA' := '1'}  				                
	SP_product_condensate_drum_low_level								: REAL;
	{attribute 'OPC.UA.DA' := '1'}  				                
	SP_product_vacuum_idle_vfd_percent									: INT;
	{attribute 'OPC.UA.DA' := '1'}  				                
	SP_product_vacuum_purge_vfd_percent									: INT;
	{attribute 'OPC.UA.DA' := '1'}  				                
	SP_product_vacuum_running_vfd_percent								: INT;
	{attribute 'OPC.UA.DA' := '1'}  				                
	SP_product_vacuum_purge_time										: REAL;							// PS 04_03_24
	{attribute 'OPC.UA.DA' := '1'}  				                
	SP_reactor_vfd_percent_maximum										: INT;
	{attribute 'OPC.UA.DA' := '1'}  				                
	SP_reactor_vfd_percent_step_duration								: REAL;
	{attribute 'OPC.UA.DA' := '1'}  				                
	SP_reactor_vfd_percent_step_size									: INT;
	{attribute 'OPC.UA.DA' := '1'}  				                
	SP_steam_bypass_duration											: REAL;
	{attribute 'OPC.UA.DA' := '1'}  				                
	SP_steam_bypass_immediately_after_warm_up							: BOOL;
	{attribute 'OPC.UA.DA' := '1'}  				                
	SP_steam_bypass_temperature											: REAL;
	{attribute 'OPC.UA.DA' := '1'}  				                
	SP_steam_bypass_vacuum_pressure										: REAL;
	{attribute 'OPC.UA.DA' := '1'}  				                
	SP_target_boiler_pressure											: REAL;
	{attribute 'OPC.UA.DA' := '1'}  				                
	SP_product_vacuum_backfeed_valve									: REAL;
	{attribute 'OPC.UA.DA' := '1'}  				                
	SP_mass_flow_totalizer												: REAL;
END_VAR

// ---- POUs/MAIN.TcPOU
PROGRAM MAIN
VAR
	bStatusListLoaded													: BOOL;
	bHalfSecondPulse													: BOOL;
	sStatusLabel														: ARRAY[0..50] OF STRING;
	tonHalfSecPulse														: TON;
END_VAR

// Phase 0 - Main
// Rev 1.0 - May 13, 2024

m01.plc_version															:= '24_05_13_02';

IF NOT bStatusListLoaded THEN
	A_Status_List();
END_IF

/// TIMER PULSE
IF tonHalfSecPulse.Q THEN
	bHalfSecondPulse													:= NOT bHalfSecondPulse;
	tonHalfSecPulse(IN:= FALSE);
END_IF
tonHalfSecPulse(IN:= TRUE, PT:= T#500MS);

P_U01();
P_M01();
P_Alarms();

ACTION A_Status_List:
// Phase 0 - A_Status_List
// Rev 1.0 - February 6, 2024

sStatusLabel[0] 														:= 'Idle';
sStatusLabel[1] 														:= '';
sStatusLabel[2]  														:= '';
sStatusLabel[3]  														:= 'Warmup running';
sStatusLabel[4]  														:= 'Steam Bypass running';
sStatusLabel[5]  														:= 'Repressurization running';
sStatusLabel[6]  														:= 'Adsorption running';
sStatusLabel[7]  														:= 'Evacuation running';
sStatusLabel[8]  														:= 'Desorption running';
sStatusLabel[9]  														:= 'Shutting down';
sStatusLabel[10]  														:= 'Pressure Test running';
sStatusLabel[11]  														:= '';
sStatusLabel[12]  														:= '';
sStatusLabel[13]  														:= 'Warmup error';
sStatusLabel[14]  														:= 'Steam Bypass error';
sStatusLabel[15]  														:= 'Repressurization error';
sStatusLabel[16]  														:= 'Adsorption error';
sStatusLabel[17]  														:= 'Evacuation error';
sStatusLabel[18]  														:= 'Desorption error';
sStatusLabel[19]  														:= 'Pressure Test error';
sStatusLabel[20]  														:= '';
sStatusLabel[21]  														:= '';
sStatusLabel[22]  														:= '';
sStatusLabel[23]  														:= 'Warmup complete';
sStatusLabel[24]  														:= 'Steam Bypass complete';
sStatusLabel[25]  														:= 'Repressurization complete';
sStatusLabel[26]  														:= 'Adsorption complete';
sStatusLabel[27]  														:= 'Evacuation complete';
sStatusLabel[28]  														:= 'Desoprtion complete';
sStatusLabel[29]  														:= 'Shutdown complete';
sStatusLabel[30]  														:= 'Pressure Test complete';
sStatusLabel[31]  														:= '';
sStatusLabel[32]  														:= 'No Reactor selected';
sStatusLabel[33]  														:= 'Stopping process';
sStatusLabel[34]  														:= 'Resetting';
sStatusLabel[35]														:= 'Saving data';
sStatusLabel[36]  														:= '';
sStatusLabel[37]  														:= '';
sStatusLabel[38]  														:= '';
sStatusLabel[39]  														:= '';
sStatusLabel[40]  														:= 'Error';
	                                    		
bStatusListLoaded														:= TRUE;
END_ACTION

END_PROGRAM

// ---- POUs/Utilities/P_U01.TcPOU
PROGRAM P_U01
VAR
	bPaul				: BOOL;
	u																	: Utility;
	
	fbWriteData															: FB_WritePersistentData;
	tonWriteData														: TON;
	bWriteData															: BOOL;
	
	sError																: STRING;
	sMessage															: STRING;
	sUtilityError														: STRING;
	sRS																	: STRING;
	iAxStep																: INT;
	i2Step																: INT;
	i3Step																: INT;
	i8Step																: INT;
	i9Step																: INT;
	iVfd_Speed															: INT;
	bAdsorptionActive													: BOOL;
	bComplete															: BOOL;
	bPreCheckDone														: BOOL;
	bTimer																: BOOL;
	bPass1																: BOOL;
	bPass2																: BOOL;
	bPass3																: BOOL;
	bPass4																: BOOL;
	bPass5																: BOOL;
	bPass6																: BOOL;
	bAdsorptionTimer													: BOOL;
	bCloseXVValves														: BOOL;
	bRunSteamBypass														: BOOL;
	bVfd_Speed_Up														: BOOL;
	rTime																: REAL;
	rSP																	: REAL;
	rPres																: REAL;
	tonTimer															: TON;
	tonAdsorptionTimer													: TON;
	tonBoilerCheck														: TON;
	
	fb_Drainage_On														: FB_Digital_Out();
	fb_Product_Condensate_Pump											: FB_Digital_Out();
	fb_Condensate_Collection_Tank_Pump									: FB_Digital_Out();
	fb_Boiler_Package													: FB_Digital_Out();
	fb_Product_Condenser												: FB_Digital_Out();
	fb_Dead_Air_Vacuum_Pump												: FB_Digital_Out();
	fb_Product_Blower													: FB_Digital_Out();
	fb_Instrument_Air_Compressor										: FB_Digital_Out();
	fb_Dead_Air_Line_C02_Pump											: FB_Digital_Out();
	fb_Dead_Air_Line_C02_Sol											: FB_Digital_Out();
	fb_Cooling_Line_Pre_Condenser_Valve									: FB_Digital_Out();
	fb_Purge_Product_Pre_Condenser_Valve								: FB_Digital_Out();
	fb_Product_Vacuum_Pump_Isolation_Valve								: FB_Digital_Out();
	fb_Product_Vacuum_Bypass_Valve										: FB_Digital_Out();
	fb_Product_Vacuum_Outlet_Isolation_Valve							: FB_Digital_Out();
	fb_Product_Condensate_Drain_Valve									: FB_Digital_Out();
	fb_Steam_Bypass_Valve												: FB_Digital_Out();
	fb_Condensate_Collection_Tank_Pump_Outlet_Valve						: FB_Digital_Out();
	fb_Product_Vacuum_Backfeed_Valve									: FB_Analog_Out();
	fb_Product_Vacuum_Backfeed_Valve_PI									: FB_PI_Control();
	fb_Product_Vacuum_Backfeed_Valve_Mode								: FB_Integer_Out();
	fb_Product_Vacuum_Pump_Vfd_Input									: FB_Analog_Out();
	fb_Product_Vacuum_Pump												: FB_Vacuum_Pump();
	fb_Product_Vacuum_Pump_Vfd											: FB_VFD();
	fb_Product_Vacuum_Pump_Radiator										: FB_Digital_Out();
	rRpm																: REAL;
	fb_Product_Blower_Vfd												: FB_VFD();
	fb_Product_Blower_Vfd_Input											: FB_Analog_Out();
	
	fb_Product_Co2_Chiller												: FB_Digital_Out();
	fb_Product_Co2_Chiller_Pump											: FB_Digital_Out();
	
	rtrigCCDrainLSHOn													: R_TRIG;
	tonCCDrainErrorOn													: TON;
	tonCCDrainErrorOff													: TON;
	bCCDrainError														: BOOL;

	rtrigPCDrainLSHOn													: R_TRIG;
	tonPCDrainErrorOn													: TON;
	tonPCDrainErrorOff													: TON;
	bPCDrainError														: BOOL;
	
	tonProductCondensatePump											: TON;
	rtrigProductCondensatePump											: R_TRIG;
	ftrigProductCondensatePump											: F_TRIG;
	bProductCondensateDrainValve										: BOOL;

	WS_Master 															: ModbusRtuMasterV2_KL6x22B;	
	WS_Errors															: MODBUS_ERRORS;
	tonWSReset															: TON;
	bWSWeather															: BOOL;
	bWSBusy																: BOOL;
	bWSError															: BOOL;
	iWSFunction															: INT;
	uiWSRead															: UINT;	
	wWSAddress															: WORD;
	wWSQuantity															: WORD;
	wWSReadData 														: ARRAY[0..21] OF WORD;
	//wWSWriteData 														: ARRAY[0..21] OF WORD;

	bBoilerOutletPresError												: BOOL;
	bBoilerOutletTempError                                              : BOOL;
	bCondensateCollectionTankFlowError									: BOOL;
	bCondensateCollectionTankLevelError									: BOOL;
	bCondensateCollectionTankO2Error									: BOOL;
	bCondensateCollectionTankOutletLineTempError                        : BOOL;
	bCondensateCollectionTankPhError									: BOOL;
	bCondensateCollectionTankTempError                                  : BOOL;
	bCondensateCollectionTankTurbidityError								: BOOL;

	bDeadAirFlowError													: BOOL;
	bDeadAirLineCo2Error												: BOOL;
	bDeadAirLinePresError												: BOOL;
	bInstrumentAirCompPresError                                         : BOOL;
	bInstrumentAirCompTempError                                         : BOOL;
	
	bPostCondenserLinePresError											: BOOL;
	bPostCondenserLineTempError                                         : BOOL;
	bPreCondenserLinePresError											: BOOL;
	bPreCondenserLineTempError                                          : BOOL;
	bProductVacuumPresError												: BOOL;
	bProductOutletPresError												: BOOL;
	bProductOutletTempError                                             : BOOL;
	bProductOutletH2oError												: BOOL;
	bProductCo2SampleH2oError											: BOOL;
	bProductOutletTemperatureError										: BOOL;
	bProductOutletCo2Error												: BOOL;
	bProductOutletO2Error												: BOOL;
	bProductOutletVolumetricFlowError									: BOOL;
	bProductOutletMassFlowError											: BOOL;
	bProductCondensateDrumLevelError									: BOOL;
	bProductCondensateValveError										: BOOL;
	bProductCondenserPumpOutlerLiquidFlowError							: BOOL;
	bProductCondenserPumpOutletTempError                                : BOOL;
	bProductVacuumPumpError												: BOOL;
	bPurgeProductLinePresError											: BOOL;
	bPurgeProductLineTempError                                          : BOOL;
	bSteamHeaderFlowError												: BOOL;
	bWaterToBoilerFlowError												: BOOL;
	bWeatherHumidityError												: BOOL;
	bWeatherPressureError												: BOOL;
	bWeatherWindSpeedError												: BOOL;
	bWeatherTempError													: BOOL;
	bWeatherTempUnsafe													: BOOL;
	bWeatherNoiseLevelError												: BOOL;
	bWeatherWindDirectionError											: BOOL;
	bSafeShutdown														: BOOL;

	sVacPumpError														: STRING;
	sVacuumPumpError													: ARRAY[0..3] OF STRING := ['', 'Cooling Temp', 'Exhaust_Temp', 'Oil_Temp'];

	// Steam Volume
	tmrTotalizers 														: TON;	
	idxSteamTable 														: INT;
	rSteamDensity 														: REAL;	
	fbSteamTotalizerEnable												: FB_Digital_Out();
END_VAR

// Phase 0 - P_U01
// Rev 1.0 - May 14, 2024

A_IO_Points();
A_Totalizers();
A_Drains();
A2_Warmup();
A3_Steam_Bypass();
A8_Shutdown();
A9_Pressure_Drop_Test();
A_BOP_Estop();
u01.shutdown_process													:= FALSE;

IF gsCycleMode = '2' THEN
	i2Step																:= 1;
	gsCycleMode															:= '';
ELSIF gsCycleMode = '3' THEN
	i3Step																:= 1;
	gsCycleMode															:= '';
ELSIF gsCycleMode = '8' THEN
	i8Step																:= 1;
	gsCycleMode															:= '';
ELSIF gsCycleMode = '9' THEN
	i9Step																:= 1;
	gsCycleMode															:= '';
END_IF

IF tonWriteData.Q OR u01.write_persistent_data THEN
	u01.write_persistent_data											:= FALSE;
	bWriteData															:= TRUE;
ELSIF NOT fbWriteData.BUSY THEN
	bWriteData															:= FALSE;
END_IF

fbWriteData(	NETID													:= '',
				PORT													:= 851,
				START													:= bWriteData,
				TMOUT													:= T#5S);

tonTimer(IN:= bTimer, PT:= REAL_TO_TIME(rTime));
tonAdsorptionTimer(IN:= bAdsorptionTimer, PT:= REAL_TO_TIME(m01.SP_adsorption_duration * _MINUTES));
tonWriteData(IN:= NOT bWriteData, PT:= T#30M);

ACTION A_BOP_Estop:
// close and stop all BOP 
IF (u.utility_error <>  '' OR P_M01_RS01.utility_error OR P_M01_RS02.utility_error OR P_M01_RS03.utility_error) 
	AND ( m01_rs1.tb_Process_Running OR  m01_rs2.tb_Process_Running OR  m01_rs3.tb_Process_Running )  THEN
	u.dead_air_vacuum_pump							:= FALSE;
	u.product_blower								:= FALSE;
	u.product_vacuum_backfeed_valve					:= _CLOSED;
	u.product_vacuum_bypass_valve					:= FALSE;
	u.product_vacuum_outlet_isolation_valve			:= FALSE;
	u.product_vacuum_pump_isolation_valve			:= FALSE;
	u.product_vacuum_pump_radiator					:= FALSE;
	u.product_vacuum_pump_vfd						:= 0;
	u.product_blower_vfd							:= 0;
	u.steam_bypass_valve							:= FALSE;
END_IF
END_ACTION

ACTION A_Drains:
// Phase 0 - P_U01.A_Drains
// Rev 1.0 - April 30, 2024

IF gbDrainageOn THEN
	
// Drain Condensate Collection Tank
	IF u.condensate_collection_tank_level > u01.SP_condensate_collection_tank_high_level THEN
		u.condensate_collection_tank_pump								:= TRUE;
		u.condensate_collection_tank_pump_outlet_valve					:= TRUE;
	END_IF
	IF u.condensate_collection_tank_level < u01.SP_condensate_collection_tank_low_level THEN
		u.condensate_collection_tank_pump								:= FALSE;
		u.condensate_collection_tank_pump_outlet_valve					:= FALSE;
	END_IF
	
	rtrigCCDrainLSHOn(CLK:= tonCCDrainErrorOn.Q);
	IF rtrigCCDrainLSHOn.Q THEN
		P_Alarms.M_Add_Alarm(_U01, gsCondensateCollectionDrainError, gsProcessStopsAtEOC);
		u.condensate_collection_tank_pump								:= FALSE;
		u.condensate_collection_tank_pump_outlet_valve					:= FALSE;
		bCCDrainError													:= TRUE;
		m01.tb_Cancel_Cycle												:= TRUE;											// Complete current cycle
	END_IF
	tonCCDrainErrorOn(IN:= u.condensate_collection_tank_lsh AND NOT bCCDrainError, PT:= _DRAIN_TIME);
	
	IF tonCCDrainErrorOff.Q THEN
		bCCDrainError													:= FALSE;
	END_IF
	tonCCDrainErrorOff(IN:= NOT u.condensate_collection_tank_lsh AND bCCDrainError, PT:= _DRAIN_TIME);
	
	
// Drain Product Condensate
	IF u.product_vacuum_pres < u01.SP_drainage_function_cutoff_pressure THEN
		u.product_condensate_pump										:= FALSE;
	ELSE
		IF u.product_condensate_drum_level > u01.SP_product_condensate_drum_high_level THEN
			u.product_condensate_pump									:= TRUE;
		END_IF
		IF u.product_condensate_drum_level < u01.SP_product_condensate_drum_low_level THEN
			u.product_condensate_pump									:= FALSE;
		END_IF
	END_IF
	
	rtrigPCDrainLSHOn(CLK:= tonPCDrainErrorOn.Q);
	IF rtrigPCDrainLSHOn.Q THEN
		P_Alarms.M_Add_Alarm(_U01, gsProductCondensateDrainError, gsProcessStopsAtEOA);
		u.product_condensate_pump										:= FALSE;
		bPCDrainError													:= TRUE;
		m01.tb_Cancel_Cycle												:= TRUE;											// Cancels all reactor sets
	END_IF
	tonPCDrainErrorOn(IN:= u.product_condensate_drum_lsh AND NOT bPCDrainError, PT:= _DRAIN_TIME);
	
	IF tonPCDrainErrorOff.Q THEN
		bPCDrainError													:= FALSE;
	END_IF
	tonPCDrainErrorOff(IN:= NOT u.product_condensate_drum_lsh AND bPCDrainError, PT:= _DRAIN_TIME);
	
END_IF
END_ACTION

ACTION A_IO_Points:
// Phase 0 - P_U01.A_IO_Points
// Rev 1.0 - May 14, 2024

// u01.point is typically from HMI or Utility programs while u.point is typically from Reactor Set through the Utility Structure.

fb_Drainage_On(Input1:= u01.drainage_on, Input2:= u.drainage_on);
gbDrainageOn															:= (u.drainage_on AND NOT u01.drainage_function_off_or) OR u01.drainage_function_on_or;

u.product_condensate_drum_lsl											:= u01.product_condensate_drum_lsl;
u.product_condensate_drum_lsh											:= u01.product_condensate_drum_lsh;
u.condensate_collection_tank_lsl										:= u01.condensate_collection_tank_lsl;
u.condensate_collection_tank_lsh										:= u01.condensate_collection_tank_lsh;

fb_Boiler_Package(Input1:= u01.boiler_package, Input2:= u.boiler_package);
u01.B_01																:= u.boiler_package;
u01.boiler_package_cmd_status											:= u.boiler_package;

// Product Condensate pump / Valve interlock & error handling
fb_Product_Condensate_Pump(Input1:= u01.product_condensate_pump, Input2:= u.product_condensate_pump);														// Get pump inputs
u01.product_condensate_pump_cmd_status									:= u.product_condensate_pump;													// Set command status (may not reflect actual output
u01.P_03																:= u.product_condensate_pump AND u01.product_condensate_drain_valve_open;		// Start pump only if on and valve is open
rtrigProductCondensatePump(CLK:= u.product_condensate_pump);
IF rtrigProductCondensatePump.Q THEN																													// Pump signal to start
	bProductCondensateValveError										:= FALSE;																		// Clear any error
	u.product_condensate_drain_valve									:= TRUE;																		// Open valve
END_IF
ftrigProductCondensatePump(CLK:= u.product_condensate_pump);
IF ftrigProductCondensatePump.Q THEN																													// Pump signal to stop
	u.product_condensate_drain_valve									:= FALSE;																		// Close valve (pump would have aleady stopped
END_IF
IF tonProductCondensatePump.Q THEN 																														// Timer has timed out (valve has not opened)
	u.product_condensate_pump											:= FALSE;																		// Turn off pump
	u.product_condensate_drain_valve									:= FALSE;																		// Close valve
	bProductCondensateValveError										:= TRUE;																		// Set holding error (keeps alarm from constantly repeating)
	P_Alarms.M_Add_Alarm(_U01, gsProductCondensateDrainValveError, gsSystemCannotRun);																	// Publish alarm
END_IF
tonProductCondensatePump(IN:= u.product_condensate_pump AND NOT u01.product_condensate_drain_valve_open, PT:= _PRODUCT_CONDENSATE_VALVE_TIME);			// Timer is on if pump on signal is true and valve is not open

fb_Product_Condensate_Drain_Valve(Input1:= u01.product_condensate_drain_valve, Input2:= u.product_condensate_drain_valve, Output=> bProductCondensateDrainValve);
u01.product_condensate_drain_valve_open_cmd_status						:= bProductCondensateDrainValve;
u01.XV_06																:= SEL(u01.P_03, bProductCondensateDrainValve, TRUE);							// Valve cannot be closed if pump is running

fb_Condensate_Collection_Tank_Pump(Input1:= u01.condensate_collection_tank_pump, Input2:= u.condensate_collection_tank_pump);
u01.P_04																:= u.condensate_collection_tank_pump;
u01.condensate_collection_tank_pump_cmd_status							:= u.condensate_collection_tank_pump;

fb_Product_Condenser(Input1:= u01.product_condenser, Input2:= u.product_condenser);
u01.E_01																:= u.product_condenser;
u01.product_condenser_cmd_status										:= u.product_condenser;

fb_Dead_Air_Vacuum_Pump(Input1:= u01.dead_air_vacuum_pump, Input2:= u.dead_air_vacuum_pump);
u01.P_01																:= u.dead_air_vacuum_pump;
u01.dead_air_vacuum_pump_cmd_status										:= u.dead_air_vacuum_pump;

fb_Product_Blower(Input1:= u01.product_blower, Input2:= u.product_blower);
u01.K_01																:= u.product_blower;
u01.product_blower_cmd_status											:= u.product_blower;

fb_Product_Blower_Vfd_Input(Input1:= u01.product_blower_vfd, Input2:= u.product_blower_vfd);
rRpm																	:= u.product_blower_vfd * _BLOWER_RPM_FACTOR;
fb_Product_Blower_Vfd(	Enable_Vfd						:= NOT u01.product_blower_vfd_ecat_state AND u01.product_blower_vfd_enable,
						Fault_Reset						:= u01.product_blower_vfd_reset,
						Rpm								:= rRpm,
						Minimum_Speed					:= _BLOWER_RPM_FACTOR * 20,
						Maximum_Speed					:= _BLOWER_RPM_FACTOR * 100, 
						StatusWord						:= u01.product_blower_vfd_status,
						ControlWord						=> u01.product_blower_vfd_control, 
						TargetRpm						=> u01.product_blower_vfd_target_vel, 
						Ready							=> u01.product_blower_vfd_enabled,
						Error							=> u01.product_blower_vfd_error);
u01.product_blower_vfd_output  									:= WORD_TO_REAL(u01.product_blower_vfd_velocity) / _BLOWER_RPM_FACTOR ;                             
//u.product_blower_vfd_output										:= WORD_TO_REAL(u01.product_blower_vfd_velocity);
IF u01.product_blower_vfd_reset THEN
	u01.product_blower_vfd_reset := FALSE;
END_IF


fb_Product_Co2_Chiller(Input1 := u01.product_co2_chiller, Input2 := u.product_co2_chiller);
u01.AT_04_chiller := u.product_co2_chiller;
u01.product_co2_chiller_cmd_status := u.product_co2_chiller;


fb_Product_Co2_Chiller_Pump(Input1 := u01.product_co2_chiller_pump, Input2 := u.product_co2_chiller_pump);
u01.AT_04_pump := u.product_co2_chiller_pump;
u01.product_co2_chiller_pump_cmd_status := u.product_co2_chiller_pump;




fb_Instrument_Air_Compressor(Input1:= u01.instrument_air_compressor, Input2:= u.instrument_air_compressor);
u01.C_01																:= u.instrument_air_compressor;
u01.instrument_air_compressor_cmd_status								:= u.instrument_air_compressor;

fb_Dead_Air_Line_C02_Pump(Input1:= u01.dead_air_line_co2_pump, Input2:= u.dead_air_line_co2_pump);
u01.AT_01_pump															:= u.dead_air_line_co2_pump;
u01.dead_air_line_co2_pump_cmd_status									:= u.dead_air_line_co2_pump;

fb_Dead_Air_Line_C02_Sol(Input1:= u01.dead_air_line_co2_sol, Input2:= u.dead_air_line_co2_sol);	
u01.AT_01_sol															:= u.dead_air_line_co2_sol;
u01.dead_air_line_co2_sol_cmd_status									:= u.dead_air_line_co2_sol;

u01.dead_air_line_co2													:= F_AnalogIn(u01.AT_01, u01.dead_air_line_co2_low, u01.dead_air_line_co2_high, u01.dead_air_line_co2_min, u01.dead_air_line_co2_offset);
u.dead_air_line_co2														:= u01.dead_air_line_co2;
u.dead_air_line_co2_error												:= u01.dead_air_line_co2_error AND NOT _DeadAirLineCo2Off;
bDeadAirLineCo2Error													:= P_Alarms.M_Check_Error(u.dead_air_line_co2_error, bDeadAirLineCo2Error, _U01, gsDeadAirLineCo2SensorError, gsProcessCannotRun);

u01.product_outlet_co2													:= F_AnalogIn(u01.AT_02A, u01.product_outlet_co2_low, u01.product_outlet_co2_high, u01.product_outlet_co2_min, u01.product_outlet_co2_offset);
u.product_outlet_co2													:= u01.product_outlet_co2;
u.product_outlet_co2_error												:= u01.product_outlet_co2_error AND NOT _ProductOutletCo2Off;
bProductOutletCo2Error													:= P_Alarms.M_Check_Error(u.product_outlet_co2_error, bProductOutletCo2Error, _U01, gsProductOutletCo2SensorError, gsProcessCannotRun);

u01.product_co2sample_h2o												:= F_AnalogIn(u01.AT_02B, u01.product_co2sample_h2o_low, u01.product_co2sample_h2o_high, u01.product_co2sample_h2o_min, u01.product_co2sample_h2o_offset);
u.product_co2sample_h2o													:= u01.product_co2sample_h2o;
u.product_co2sample_h2o_error											:= u01.product_co2sample_h2o_error AND NOT _ProductCo2SampleH2oOff;
bProductCo2SampleH2oError												:= P_Alarms.M_Check_Error(u.product_co2sample_h2o_error, bProductCo2SampleH2oError, _U01, gsProductCo2SampleH2oSensorError, gsProcessCannotRun);

u01.product_outlet_h2o													:= F_AnalogIn(u01.AT_07A, u01.product_outlet_h2o_low, u01.product_outlet_h2o_high, u01.product_outlet_h2o_min, u01.product_outlet_h2o_offset);
u.product_outlet_h2o													:= u01.product_outlet_h2o;
u.product_outlet_h2o_error												:= u01.product_outlet_h2o_error AND NOT _ProductOutletH2oOff;
bProductOutletH2oError													:= P_Alarms.M_Check_Error(u.product_outlet_h2o_error, bProductOutletH2oError, _U01, gsProductOutletH2oSensorError, gsProcessCannotRun);

u01.product_outlet_temperature											:= F_AnalogIn(u01.AT_07B, u01.product_outlet_temperature_low, u01.product_outlet_temperature_high, u01.product_outlet_temperature_min, u01.product_outlet_temperature_offset);
u.product_outlet_temperature											:= u01.product_outlet_temperature;
u.product_outlet_temperature_error										:= u01.product_outlet_temperature_error AND NOT _ProductOutletTemperatureOff;
bProductOutletTemperatureError											:= P_Alarms.M_Check_Error(u.product_outlet_temperature_error, bProductOutletTemperatureError, _U01, gsProductOutletTemperatureSensorError, gsProcessCannotRun);

u01.product_outlet_o2													:= F_AnalogIn(u01.AT_03, u01.product_outlet_o2_low, u01.product_outlet_o2_high, u01.product_outlet_o2_min, u01.product_outlet_o2_offset);
u.product_outlet_o2														:= u01.product_outlet_o2;
u.product_outlet_o2_error												:= u01.product_outlet_o2_error AND NOT _ProductOutletO2Off;
bProductOutletO2Error													:= P_Alarms.M_Check_Error(u.product_outlet_o2_error, bProductOutletO2Error, _U01, gsProductOutletO2SensorError, gsProcessCannotRun);




u01.condensate_collection_tank_ph										:= F_AnalogIn(u01.AT_04, u01.condensate_collection_tank_ph_low, u01.condensate_collection_tank_ph_high, u01.condensate_collection_tank_ph_min, u01.condensate_collection_tank_ph_offset);
u.condensate_collection_tank_ph											:= u01.condensate_collection_tank_ph;
u.condensate_collection_tank_ph_error									:= u01.condensate_collection_tank_ph_error AND NOT _CondensateCollectionTankPhOff;
bCondensateCollectionTankPhError										:= P_Alarms.M_Check_Error(u.condensate_collection_tank_ph_error, bCondensateCollectionTankPhError, _U01, gsCondensateCollectionTankPhSensorError, gsProcessCannotRun);

u01.condensate_collection_tank_o2										:= F_AnalogIn(u01.AT_05, u01.condensate_collection_tank_o2_low, u01.condensate_collection_tank_o2_high, u01.condensate_collection_tank_o2_min, u01.condensate_collection_tank_o2_offset);
u.condensate_collection_tank_o2											:= u01.condensate_collection_tank_o2;
u.condensate_collection_tank_o2_error									:= u01.condensate_collection_tank_o2_error AND NOT _CondensateCollectionTankO2Off;
bCondensateCollectionTankO2Error										:= P_Alarms.M_Check_Error(u.condensate_collection_tank_o2_error, bCondensateCollectionTankO2Error, _U01, gsCondensateCollectionTankO2SensorError, gsProcessCannotRun);

u01.condensate_collection_tank_turbidity								:= F_AnalogIn(u01.AT_06, u01.condensate_collection_tank_turbidity_low, u01.condensate_collection_tank_turbidity_high, u01.condensate_collection_tank_turbidity_min, u01.condensate_collection_tank_turbidity_offset);
u.condensate_collection_tank_turbidity									:= u01.condensate_collection_tank_turbidity;
u.condensate_collection_tank_turbidity_error							:= u01.condensate_collection_tank_turbidity_error AND NOT _CondensateCollectionTankTurbidityOff;
bCondensateCollectionTankTurbidityError									:= P_Alarms.M_Check_Error(u.condensate_collection_tank_turbidity_error, bCondensateCollectionTankTurbidityError, _U01, gsCondensateCollectionTankTurbiditySensorError, gsProcessCannotRun);

u01.weather_humidity													:= F_AnalogIn(u01.AT_07, u01.weather_humidity_low, u01.weather_humidity_high, u01.weather_humidity_min, u01.weather_humidity_offset);
u.weather_humidity														:= u01.weather_humidity;
u.weather_humidity_error												:= u01.weather_humidity_error AND NOT _WeatherHumidityOff;
bWeatherHumidityError													:= P_Alarms.M_Check_Error(u.weather_humidity_error, bWeatherHumidityError, _U01, gsWeatherHumiditySensorError, gsProcessCannotRun);

u01.weather_pres														:= F_AnalogIn(u01.PT_09, u01.weather_pres_low, u01.weather_pres_high, u01.weather_pres_min, u01.weather_pres_offset);
u.weather_pres															:= u01.weather_pres;
u.weather_pres_error													:= u01.weather_pres_error AND NOT _WeatherPressureOff;
bWeatherPressureError													:= P_Alarms.M_Check_Error(u.weather_pres_error, bWeatherPressureError, _U01, gsWeatherPresureSensorError, gsProcessCannotRun);

u01.weather_wind_speed													:= F_AnalogIn(u01.AT_08, u01.weather_wind_speed_low, u01.weather_wind_speed_high, u01.weather_wind_speed_min, u01.weather_wind_speed_offset);
u.weather_wind_speed													:= u01.weather_wind_speed;
u.weather_wind_speed_error												:= u01.weather_wind_speed_error AND NOT _WeatherWindSpeedOff;
bWeatherWindSpeedError													:= P_Alarms.M_Check_Error(u.weather_wind_speed_error, bWeatherWindSpeedError, _U01, gsWeatherWindSpeedSensorError, gsProcessCannotRun);

u01.weather_temp														:= F_Temperature(u01.TT_10, u01.weather_temp_offset);
u.weather_temp															:= u01.weather_temp;
u.weather_temp_error													:= u01.weather_temp_error AND NOT _WeatherTempOff;
bWeatherTempError														:= P_Alarms.M_Check_Error(u.weather_temp_error, bWeatherTempError, _U01, gsWeatherTempSensorError, gsProcessCannotRun);
IF u.weather_temp > m01.SP_maximum_inlet_air_temperature_during_adsorption OR u.weather_temp < m01.SP_minimum_inlet_air_temperature_during_adsorption THEN
	u.os_air_unsafe_temp												:= TRUE;
ELSIF u.weather_temp <= m01.SP_maximum_inlet_air_temperature_during_adsorption - _TEMP_DEADBAND AND u.weather_temp >= m01.SP_minimum_inlet_air_temperature_during_adsorption + _TEMP_DEADBAND THEN
	u.os_air_unsafe_temp												:= FALSE;
END_IF
bWeatherTempUnsafe														:= P_Alarms.M_Check_Error(u.os_air_unsafe_temp, bWeatherTempUnsafe, _U01, gsOutsideTempRangeError, gsSystemCannotRun);

u01.weather_noise_level													:= F_AnalogIn(u01.NT_01, 0, 100, 0, 0);
u.weather_noise_level													:= u01.weather_noise_level;
u.weather_noise_level_error												:= u01.weather_noise_level_error AND NOT _WeatherNoiseLevelOff;
bWeatherNoiseLevelError													:= P_Alarms.M_Check_Error(u.weather_noise_level_error, bWeatherNoiseLevelError, _U01, gsWeatherNoiseLevelSensorError, gsProcessCannotRun);

u01.weather_wind_direction												:= F_AnalogIn(u01.WDT_01, 0, 100, 0, 0);
u.weather_wind_direction												:= u01.weather_wind_direction;
u.weather_wind_direction_error											:= u01.weather_wind_direction_error AND NOT _WeatherWindDirectionOff;
bWeatherWindDirectionError												:= P_Alarms.M_Check_Error(u.weather_wind_direction_error, bWeatherWindDirectionError, _U01, gsWeatherWindDirectionSensorError, gsProcessCannotRun);

u01.dead_air_flow														:= F_AnalogIn(u01.FT_01, u01.dead_air_flow_low, u01.dead_air_flow_high, u01.dead_air_flow_min, u01.dead_air_flow_offset);
u.dead_air_flow															:= u01.dead_air_flow;
u.dead_air_flow_error													:= u01.dead_air_flow_error AND NOT _DeadAirFlowOff;
bDeadAirFlowError														:= P_Alarms.M_Check_Error(u.dead_air_flow_error, bDeadAirFlowError, _U01, gsDeadAirFlowSensorError, gsProcessCannotRun);

u01.product_outlet_volumetric_flow										:= F_AnalogIn(u01.FT_03, u01.product_outlet_volumetric_flow_low, u01.product_outlet_volumetric_flow_high, u01.product_outlet_volumetric_flow_min, u01.product_outlet_volumetric_flow_offset);
u.product_outlet_volumetric_flow										:= u01.product_outlet_volumetric_flow;
u.product_outlet_volumetric_flow_error									:= u01.product_outlet_volumetric_flow_error AND NOT _ProductOutVolumetricFlowOff;
bProductOutletVolumetricFlowError										:= P_Alarms.M_Check_Error(u.product_outlet_volumetric_flow_error, bProductOutletVolumetricFlowError, _U01, gsProductOutletVolumetricFlowSensorError, gsProcessCannotRun);

u01.product_outlet_mass_flow											:= F_AnalogIn(u01.FT_02, u01.product_outlet_mass_flow_low, u01.product_outlet_mass_flow_high, u01.product_outlet_mass_flow_min, u01.product_outlet_mass_flow_offset);
u.product_outlet_mass_flow												:= u01.product_outlet_mass_flow;
u.product_outlet_mass_flow_error										:= u01.product_outlet_mass_flow_error AND NOT _ProductOutMassFlowOff;
bProductOutletMassFlowError												:= P_Alarms.M_Check_Error(u.product_outlet_mass_flow_error, bProductOutletMassFlowError, _U01, gsProductOutletMassFlowSensorError, gsProcessCannotRun);

u01.product_condenser_pump_outlet_liquid_flow							:= F_AnalogIn(u01.FT_04, u01.product_condenser_pump_outlet_liquid_flow_low, u01.product_condenser_pump_outlet_liquid_flow_high, u01.product_condenser_pump_outlet_liquid_flow_min, u01.product_condenser_pump_outlet_liquid_flow_offset);
u.product_condenser_pump_outlet_liquid_flow								:= u01.product_condenser_pump_outlet_liquid_flow;
u.product_condenser_pump_outlet_liquid_flow_error						:= u01.product_condenser_pump_outlet_liquid_flow_error AND NOT _ProductCondenserPumpOutlerLiquidFlowOff;
bProductCondenserPumpOutlerLiquidFlowError								:= P_Alarms.M_Check_Error(u.product_condenser_pump_outlet_liquid_flow_error, bProductCondenserPumpOutlerLiquidFlowError, _U01, gsProductCondenserPumpOutletLiquidFlowSensorError, gsProcessCannotRun);
	
u01.tap_water_to_boiler_flow											:= F_AnalogIn(u01.FT_05, u01.tap_water_to_boiler_flow_low, u01.tap_water_to_boiler_flow_high, u01.tap_water_to_boiler_flow_min, u01.tap_water_to_boiler_flow_offset);
u.tap_water_to_boiler_flow												:= u01.tap_water_to_boiler_flow;
u.tap_water_to_boiler_flow_error										:= u01.tap_water_to_boiler_flow_error AND NOT _WaterToBoilerFlowOff;
bWaterToBoilerFlowError													:= P_Alarms.M_Check_Error(u.tap_water_to_boiler_flow_error, bWaterToBoilerFlowError, _U01, gsTapWaterToBoilerFlowSensorError, gsProcessCannotRun);

u01.steam_header_flow													:= F_AnalogIn(u01.FT_06, u01.steam_header_flow_low, u01.steam_header_flow_high, u01.steam_header_flow_min, u01.steam_header_flow_offset);
u.steam_header_flow														:= u01.steam_header_flow;
u.steam_header_flow_error												:= u01.steam_header_flow_error AND NOT _SteamHeadFlowOff;
bSteamHeaderFlowError													:= P_Alarms.M_Check_Error(u.steam_header_flow_error, bSteamHeaderFlowError, _U01, gsSteamHeaderFlowSensorError, gsProcessCannotRun);
	
u01.condensate_collection_tank_flow										:= F_AnalogIn(u01.FT_07, u01.condensate_collection_tank_flow_low, u01.condensate_collection_tank_flow_high, u01.condensate_collection_tank_flow_min, u01.condensate_collection_tank_flow_offset);
u.condensate_collection_tank_flow										:= u01.condensate_collection_tank_flow;
u.condensate_collection_tank_flow_error									:= u01.condensate_collection_tank_flow_error AND NOT _CondensateCollectionTankFlowOff;
bCondensateCollectionTankFlowError										:= P_Alarms.M_Check_Error(u.condensate_collection_tank_flow_error, bCondensateCollectionTankFlowError, _U01, gsCondensateCollectionTankFlowSensorError, gsProcessCannotRun);
	
u01.product_condensate_drum_level										:= F_AnalogIn(u01.LT_01, u01.product_condensate_drum_level_low, u01.product_condensate_drum_level_high, u01.product_condensate_drum_level_min, u01.product_condensate_drum_level_offset);
u.product_condensate_drum_level											:= u01.product_condensate_drum_level;
u.product_condensate_drum_level_error									:= u01.product_condensate_drum_level_error AND NOT _ProductCondensateDrumLevelOff;
bProductCondensateDrumLevelError										:= P_Alarms.M_Check_Error(u.product_condensate_drum_level_error, bProductCondensateDrumLevelError, _U01, gsProductCondensateDrumLevelSensorError, gsProcessCannotRun);
	
u01.condensate_collection_tank_level									:= F_AnalogIn(u01.LT_02, u01.condensate_collection_tank_level_low, u01.condensate_collection_tank_level_high, u01.condensate_collection_tank_level_min, u01.condensate_collection_tank_level_offset);
u.condensate_collection_tank_level										:= u01.condensate_collection_tank_level;
u.condensate_collection_tank_level_error								:= u01.condensate_collection_tank_level_error AND NOT _CondensateCollectionTankLevelOff;
bCondensateCollectionTankLevelError										:= P_Alarms.M_Check_Error(u.condensate_collection_tank_level_error, bCondensateCollectionTankLevelError, _U01, gsCondensateCollectionTankLevelSensorError, gsProcessCannotRun);
	
u01.dead_air_line_pres													:= F_AnalogIn(U01.PT_01, u01.dead_air_line_pres_low, u01.dead_air_line_pres_high, u01.dead_air_line_pres_min, u01.dead_air_line_pres_offset);
u.dead_air_line_pres													:= u01.dead_air_line_pres;
u.dead_air_line_pres_error												:= u01.dead_air_line_pres_error AND NOT _DeadAirLinePresOff;
bDeadAirLinePresError													:= P_Alarms.M_Check_Error(u.dead_air_line_pres_error, bDeadAirLinePresError, _U01, gsDeadAirLinePresSensorError, gsProcessCannotRun);

u01.purge_product_line_pres												:= F_AnalogIn(U01.PT_02, u01.purge_product_line_pres_low, u01.purge_product_line_pres_high, u01.purge_product_line_pres_min, u01.purge_product_line_pres_offset);
u.purge_product_line_pres												:= u01.purge_product_line_pres;
u.purge_product_line_pres_error											:= u01.purge_product_line_pres_error AND NOT _PurgeProductLinePresOff;
bPurgeProductLinePresError												:= P_Alarms.M_Check_Error(u.purge_product_line_pres_error, bPurgeProductLinePresError, _U01, gsPurgeProductLinePresSensorError, gsProcessCannotRun);

u01.pre_condenser_line_pres												:= F_AnalogIn(U01.PT_03, u01.pre_condenser_line_pres_low, u01.pre_condenser_line_pres_high, u01.pre_condenser_line_pres_min, u01.pre_condenser_line_pres_offset);
u.pre_condenser_line_pres												:= u01.pre_condenser_line_pres;
u.pre_condenser_line_pres_error											:= u01.pre_condenser_line_pres_error AND NOT _PreCondenserLinePresOff;
bPreCondenserLinePresError												:= P_Alarms.M_Check_Error(u.pre_condenser_line_pres_error, bPreCondenserLinePresError, _U01, gsPreCondenserLinePresSensorError, gsProcessCannotRun);

u01.post_condenser_line_pres											:= F_AnalogIn(U01.PT_04, u01.post_condenser_line_pres_low, u01.post_condenser_line_pres_high, u01.post_condenser_line_pres_min, u01.post_condenser_line_pres_offset);
u.post_condenser_line_pres												:= u01.post_condenser_line_pres;
u.post_condenser_line_pres_error										:= u01.post_condenser_line_pres_error AND NOT _PostCondenserLinePresOff;
bPostCondenserLinePresError												:= P_Alarms.M_Check_Error(u.post_condenser_line_pres_error, bPostCondenserLinePresError, _U01, gsPostCondenserLinePresSensorError, gsProcessCannotRun);

u01.product_vacuum_pres													:= F_AnalogIn(U01.PT_05, u01.product_vacuum_pres_low, u01.product_vacuum_pres_high, u01.product_vacuum_pres_min, u01.product_vacuum_pres_offset);
u.product_vacuum_pres													:= u01.product_vacuum_pres;
u.product_vacuum_pres_error												:= u01.product_vacuum_pres_error AND NOT _ProductVacuumPresOff;
bProductVacuumPresError													:= P_Alarms.M_Check_Error(u.product_vacuum_pres_error, bProductVacuumPresError, _U01, gsProductVacuumPresSensorError, gsProcessCannotRun);

u01.product_outlet_pres													:= F_AnalogIn(U01.PT_06, u01.product_outlet_pres_low, u01.product_outlet_pres_high, u01.product_outlet_pres_min, u01.product_outlet_pres_offset);
u.product_outlet_pres													:= u01.product_outlet_pres;
u.product_outlet_pres_error												:= u01.product_outlet_pres_error AND NOT _ProductOutletPresOff;
bProductOutletPresError													:= P_Alarms.M_Check_Error(u.product_outlet_pres_error, bProductOutletPresError, _U01, gsProductOutletPresSensorError, gsProcessCannotRun);

u01.boiler_outlet_pres													:= F_AnalogIn(U01.PT_07, u01.boiler_outlet_pres_low, u01.boiler_outlet_pres_high, u01.boiler_outlet_pres_min, u01.boiler_outlet_pres_offset);
u.boiler_outlet_pres													:= u01.boiler_outlet_pres;
u.boiler_outlet_pres_error												:= u01.boiler_outlet_pres_error AND NOT _BoilerOutletPresOff;
bBoilerOutletPresError													:= P_Alarms.M_Check_Error(u.boiler_outlet_pres_error, bBoilerOutletPresError, _U01, gsBoilerOutletPresSensorError, gsProcessCannotRun);

u01.purge_product_line_temp												:= F_Temperature(u01.TT_01, u01.purge_product_line_temp_offset);
u.purge_product_line_temp												:= u01.purge_product_line_temp;
u.purge_product_line_temp_error											:= u01.purge_product_line_temp_error AND NOT _PurgeProductLineTempOff;
bPurgeProductLineTempError												:= P_Alarms.M_Check_Error(u.purge_product_line_temp_error, bPurgeProductLineTempError, _U01, gsPurgeProductLineTempSensorError, gsProcessCannotRun);

u01.pre_condenser_line_temp												:= F_Temperature(u01.TT_02, u01.pre_condenser_line_temp_offset);
u.pre_condenser_line_temp												:= u01.pre_condenser_line_temp;
u.pre_condenser_line_temp_error											:= u01.pre_condenser_line_temp_error AND NOT _PreCondenserLineTempOff;
bPreCondenserLineTempError												:= P_Alarms.M_Check_Error(u.pre_condenser_line_temp_error, bPreCondenserLineTempError, _U01, gsPreCondenserLineTempSensorError, gsProcessCannotRun);

u01.post_condenser_line_temp											:= F_Temperature(u01.TT_03, u01.post_condenser_line_temp_offset);
u.post_condenser_line_temp												:= u01.post_condenser_line_temp;
u.post_condenser_line_temp_error										:= u01.post_condenser_line_temp_error AND NOT _PostCondenserLineTempOff;
bPostCondenserLineTempError												:= P_Alarms.M_Check_Error(u.post_condenser_line_temp_error, bPostCondenserLineTempError, _U01, gsPostCondenserLineTempSensorError, gsProcessCannotRun);
	
u01.product_outlet_temp													:= F_Temperature(u01.TT_04, u01.product_outlet_temp_offset);
u.product_outlet_temp													:= u01.product_outlet_temp;
u.product_outlet_temp_error												:= u01.product_outlet_temp_error AND NOT _ProductOutletTempOff;
bProductOutletTempError													:= P_Alarms.M_Check_Error(u.product_outlet_temp_error, bProductOutletTempError, _U01, gsProductOutletTempSensorError, gsProcessCannotRun);
	
u01.product_condenser_pump_outlet_temp									:= F_Temperature(u01.TT_05, u01.product_condenser_pump_outlet_temp_offset);
u.product_condenser_pump_outlet_temp									:= u01.product_condenser_pump_outlet_temp;
u.product_condenser_pump_outlet_temp_error								:= u01.product_condenser_pump_outlet_temp_error AND NOT _ProductCondenserPumpOutletTempOff;
bProductCondenserPumpOutletTempError									:= P_Alarms.M_Check_Error(u.product_condenser_pump_outlet_temp_error, bProductCondenserPumpOutletTempError, _U01, gsProductCondenserPumpOutletTempSensorError, gsProcessCannotRun);
	
u01.boiler_outlet_temp													:= F_Temperature(u01.TT_06, u01.boiler_outlet_temp_offset);
u.boiler_outlet_temp													:= u01.boiler_outlet_temp;
u.boiler_outlet_temp_error												:= u01.boiler_outlet_temp_error AND NOT _BoilerOutletTempOff;
bBoilerOutletTempError													:= P_Alarms.M_Check_Error(u.boiler_outlet_temp_error, bBoilerOutletTempError, _U01, gsBoilerOutletTempSensorError, gsProcessCannotRun);
	
u01.condensate_collection_tank_temp										:= F_Temperature(u01.TT_07, u01.condensate_collection_tank_temp_offset);
u.condensate_collection_tank_temp										:= u01.condensate_collection_tank_temp;
u.condensate_collection_tank_temp_error									:= u01.condensate_collection_tank_temp_error AND NOT _CondensateCollectionTankTempOff;
bCondensateCollectionTankTempError										:= P_Alarms.M_Check_Error(u.condensate_collection_tank_temp_error, bCondensateCollectionTankTempError, _U01, gsCondensateCollectionTankTempSensorError, gsProcessCannotRun);
	
u01.condensate_collection_tank_outlet_line_temp							:= F_Temperature(u01.TT_08, u01.condensate_collection_tank_outlet_line_temp_offset);
u.condensate_collection_tank_outlet_line_temp							:= u01.condensate_collection_tank_outlet_line_temp;
u.condensate_collection_tank_outlet_line_temp_error						:= u01.condensate_collection_tank_outlet_line_temp_error AND NOT _CondensateCollectionTankOutletLineTempOff;
bCondensateCollectionTankOutletLineTempError							:= P_Alarms.M_Check_Error(u.condensate_collection_tank_outlet_line_temp_error, bCondensateCollectionTankOutletLineTempError, _U01, gsCondensateCollectionTankOutletLineTempSensorError, gsProcessCannotRun);

u01.instrument_air_comp_pres											:= F_AnalogIn(U01.PT_08, u01.instrument_air_comp_pres_low, u01.instrument_air_comp_pres_high, u01.instrument_air_comp_pres_min, u01.instrument_air_comp_pres_offset);
u.instrument_air_comp_pres												:= u01.instrument_air_comp_pres;
u.instrument_air_comp_pres_error										:= u01.instrument_air_comp_pres_error AND NOT _InstrumentAirCompPresOff;
bInstrumentAirCompPresError												:= P_Alarms.M_Check_Error(u.instrument_air_comp_pres_error, bInstrumentAirCompPresError, _U01, gsInstrumentAirCompPresSensorError, gsProcessCannotRun);
rPres																	:= SEL(u.instrument_air_comp_pres_error, u01.instrument_air_comp_pres, -100);
IF rPres >= u01.SP_minimum_instrument_air_pressure AND rPres <= u01.SP_acceptable_low_instrument_air_pressure THEN 
	u.instrument_air_comp_pres_interlock								:= 1;
ELSIF rPres <= u01.SP_maximum_instrument_air_pressure AND rPres >= u01.SP_acceptable_high_instrument_air_pressure THEN 
	u.instrument_air_comp_pres_interlock								:= 1;
ELSIF rPres < u01.SP_minimum_instrument_air_pressure OR rPres > u01.SP_maximum_instrument_air_pressure THEN
	u.instrument_air_comp_pres_interlock								:= 2;
ELSE
	u.instrument_air_comp_pres_interlock								:= 0;
END_IF	

u01.instrument_air_comp_temp											:= F_Temperature(u01.TT_09, u01.instrument_air_comp_temp_offset);
u.instrument_air_comp_temp												:= u01.instrument_air_comp_temp;
u.instrument_air_comp_temp_error										:= u01.instrument_air_comp_temp_error AND NOT _InstrumentAirCompTempOff;

bInstrumentAirCompTempError												:= P_Alarms.M_Check_Error(u.instrument_air_comp_temp_error, bInstrumentAirCompTempError, _U01, gsInstrumentAirCompTempSensorError, gsProcessCannotRun);
IF NOT bInstrumentAirCompTempError THEN
	IF u.instrument_air_comp_temp < u01.SP_minimum_instrument_air_temperature OR u.instrument_air_comp_temp > u01.SP_maximum_instrument_air_temperature THEN
		P_Alarms.M_Add_Alarm(_U01, gsPneumaticLineTempError, gsReactorSetCannotRun);
		bInstrumentAirCompTempError										:= TRUE;
	END_IF
END_IF

IF bCloseXVValves THEN
	u01.cooling_line_pre_condenser_valve								:= FALSE;
	u01.purge_product_pre_condenser_valve								:= FALSE;
	u01.product_vacuum_pump_isolation_valve								:= FALSE;
	u01.product_vacuum_bypass_valve										:= FALSE;
	u01.product_vacuum_outlet_isolation_valve							:= FALSE;
	u01.steam_bypass_valve												:= FALSE;
	u01.condensate_collection_tank_pump_outlet_valve					:= FALSE;
	bCloseXVValves														:= FALSE;
END_IF
	
fb_Cooling_Line_Pre_Condenser_Valve(Input1:= u01.cooling_line_pre_condenser_valve, Input2:= u.cooling_line_pre_condenser_valve, Output=> u01.XV_01);
u01.cooling_line_pre_condenser_valve_open_cmd_status					:= u01.XV_01;
u.cooling_line_pre_condenser_valve_clear								:= F_ValveClear(u.cooling_line_pre_condenser_valve, u01.cooling_line_pre_condenser_valve_open, u01.cooling_line_pre_condenser_valve_closed);

fb_Purge_Product_Pre_Condenser_Valve(Input1:= u01.purge_product_pre_condenser_valve, Input2:= u.purge_product_pre_condenser_valve, Output=> u01.XV_02);
u01.purge_product_pre_condenser_valve_open_cmd_status					:= u01.XV_02;
u.purge_product_pre_condenser_valve_clear								:= F_ValveClear(u.purge_product_pre_condenser_valve, u01.purge_product_pre_condenser_valve_open, u01.purge_product_pre_condenser_valve_closed);

fb_Product_Vacuum_Pump_Isolation_Valve(Input1:= u01.product_vacuum_pump_isolation_valve, Input2:= u.product_vacuum_pump_isolation_valve, Output=> u01.XV_03);
u01.product_vacuum_pump_isolation_valve_open_cmd_status					:= u01.XV_03;
u.product_vacuum_pump_isolation_valve_clear								:= F_ValveClear(u.product_vacuum_pump_isolation_valve, u01.product_vacuum_pump_isolation_valve_open, u01.product_vacuum_pump_isolation_valve_closed);

fb_Product_Vacuum_Bypass_Valve(Input1:= u01.product_vacuum_bypass_valve, Input2:= u.product_vacuum_bypass_valve, Output=> u01.XV_04);
u01.product_vacuum_bypass_valve_open_cmd_status							:= u01.XV_04;
u.product_vacuum_bypass_valve_clear										:= F_ValveClear(u.product_vacuum_bypass_valve, u01.product_vacuum_bypass_valve_open, u01.product_vacuum_bypass_valve_closed);

